(* CODESYS project test_IMA-TECHDays
   Author: SESA697794
   DefaultNamespace: MulticarrierExample
   Title: Git_example
   Version: 0.0.0.0

Project tree, tasks and I/O mapping:
  LMC_PacDrive : PacDrive LMC 300/400/402/600/802/902C, Schneider Electric, order no. LMC Pro and Pro2, version 1.76.12.4
    application Application
      libraries: PD_PacDriveLib, 1.11.1.0 (Schneider Electric); ApplicationLogger, 1.1.7.0 (Schneider Electric); Mathematics, 1.0.4.0 (Schneider Electric); Multicarrier, 1.3.6.0 (Schneider Electric); MulticarrierStation, 1.2.0.0 (Schneider Electric); DigitalTwinCommunication, 1.2.1.0 (Schneider Electric); SercosCommunication, 1.2.4.0 (Schneider Electric); PD_SoMotionGenerator, 1.9.4.0 (Schneider Electric); SysMem, * (System); SysTime, * (System); TcpUdpCommunication, 2.3.0.0 (Schneider Electric); PD_GlobalDiagnostics, 1.6.0.0 (Schneider Electric); PD_AxisModule, 1.7.1.0 (Schneider Electric); PD_Template, 1.9.0.0 (Schneider Electric); IecRtsServices, 1.0.5.0 (Schneider Electric); VisuDialogs, * (System)
      task TASK_Communication (cyclic, interval T#20ms, priority 30) calls SR_EmulationInterface, SR_OpcUa
      task TASK_SR_Diagnostics (cyclic, interval T#100ms, priority 31, watchdog T#100ms x 2) calls SR_Diagnostics
      task TASK_SR_Logging (cyclic, interval T#10ms, priority 13, watchdog T#10ms x 2) calls SR_Logging
      task TASK_SR_MainMachine (cyclic, interval T#5ms, priority 8, watchdog T#5ms x 10) calls SR_HWCopyIO, SR_MainMachine
      task TASK_SR_SlowTask (cyclic, interval T#200ms, priority 29) calls SR_ReadControlLoopParameter, SR_WriteControlLoopParameter
      task TASK_SR_VisControl (cyclic, interval T#50ms, priority 14, watchdog T#50ms x 2) calls SR_VisControl
      Application Logger
      Check_Lib/
        function CheckBounds [ST]
        function CheckDivDInt [ST]
        function CheckDivLInt [ST]
        function CheckDivLReal [ST]
        function CheckDivReal [ST]
        function CheckPointer [ST]
        function CheckRangeSigned [ST]
        function CheckRangeUnsigned [ST]
      MulticarrierConfiguration
      MulticarrierConfiguration/
        global variables GVL_MulticarrierConfiguration
        data type ST_Carrier
        data type ST_CarrierCompound
        data type ST_CarrierType
        data type ST_Part
        data type ST_PartType
        data type ST_Physics
        data type ST_ProductType
        data type ST_Segment
        data type ST_SegmentType
        data type ST_Station
        data type ST_ToolType
        data type ST_Track
      MulticarrierEmulation/
        global variables GVL_MulticarrierEmulation
        program SR_EmulationInterface [ST]: Init_MulticarrierEmulation
        Symbol Configuration
      ParameterListCarrier
      ParameterListSegments
      TemplateFullProgrammingFramework/
        CamDiagram_Slave1
          Segment
          Segment
          Segment
        CamDiagram_Slave2
          Segment
          Segment
          Segment
        EquipmentModules/
          MulticarrierModule/
            data type ET_OpModeVis
            data type ET_TraceSource
            data type ET_VisPosGapDist
            function FC_LrealEqual [ST]
            function FC_SplitString [ST]
            Multicarrier Stations/
              AutomaticMode/
                Base Station/
                  data type ET_ResultSource
                  data type ET_ResultStation
                  data type ET_StationType
                function block FB_Station1 [ST]: CyclicMotionCall
                visualisation Vis_Auto
                visualisation Vis_StationCopyMaster
              data type ST_StationParameter
              Test Multicarrier/
                01_PlayGround/
                  Traces/
                  Vis_MoveCmds/
                02_SimpleStation/
                03_PosAndSync/
                04_ColorStations/
                05_VelLimitStation/
                06_StandardStations/
                07_ExternalMaster/
                08_Superimpose/
                function block FB_MotionTestStationBase [ST]
                program SR_CallTestStations [ST]
                data type ST_CarrierMotionData
                data type ST_EmulationTestStations
                visualisation Vis_TestMulticarrier
            program SR_CarriersInStationToTrace [ST]: Call
            program SR_MulticarrierModule [SFC]: Init_CmdTables, Init_SubModules, ControlEnable, ControlModule, AddMessageToAPL, APLStartPosEndPos, TraceAndAPL, TraceStartPosEndPos, ExceptionControl_Action, HardwareFaults, Init_Exceptions, Init_Reactions, ModuleFaults, StopAllCarriers, ExitLastOpMode, MoveAllCarriersInFirstStation, SetMinGapForMoveGapControl, VirtualSetPosOfAllCarriers, Init_Carriers, Init_CrashPrevention, Init_FeedbackForVis, Init_Track, InitModule_Action, Manual_Entry, Manual_Exit, Manual_Logic, RegisterLoggerPoint, CallAllStations, DeleteAllCarriersFromStations, ErrorQuitStations, ErrorsFromStations, Init_RegisterStationsToAPL, ParameterStation1, ParameterStation2, SetStationTriggerViaTimer, TraceStations, StoreCurrentMoveCmds, Input_Action, Logger_Action, Logic_active, Output_Active, Start_Action, SubModules_Action, UpdateStructs, TrackCalibration_Logic
            data type ST_MulticarrierModule
            Traces/
              trace Trace_PosVelAcc_CurrentTrackDeviation (task SystemMotionTask): SR_MulticarrierModule.aifTraceObject[1].udiCarrierIndex, SR_MulticarrierModule.aifTraceObject[1].ifFeedbackMotionValues.lrRefTrackPosition, SR_MulticarrierModule.aifTraceObject[1].ifFeedbackMotionValues.lrRefVelocity, SR_MulticarrierModule.aifTraceObject[1].ifFeedbackMotionValues.lrRefAcceleration, SR_MulticarrierModule.aifTraceCarrierMovementData[1].ActualCurrent, SR_MulticarrierModule.aifTraceCarrierMovementData[1].TrackingDeviation, SR_MulticarrierModule.aifTraceObject[2].udiCarrierIndex, SR_MulticarrierModule.aifTraceObject[2].ifFeedbackMotionValues.lrRefTrackPosition, SR_MulticarrierModule.aifTraceObject[2].ifFeedbackMotionValues.lrRefVelocity, SR_MulticarrierModule.aifTraceObject[2].ifFeedbackMotionValues.lrRefAcceleration, SR_MulticarrierModule.aifTraceCarrierMovementData[2].ActualCurrent, SR_MulticarrierModule.aifTraceCarrierMovementData[2].TrackingDeviation, SR_MulticarrierModule.aifTraceObject[3].udiCarrierIndex, SR_MulticarrierModule.aifTraceObject[3].ifFeedbackMotionValues.lrRefTrackPosition, SR_MulticarrierModule.aifTraceObject[3].ifFeedbackMotionValues.lrRefVelocity, SR_MulticarrierModule.aifTraceObject[3].ifFeedbackMotionValues.lrRefAcceleration, SR_MulticarrierModule.aifTraceCarrierMovementData[3].ActualCurrent, SR_MulticarrierModule.aifTraceCarrierMovementData[3].TrackingDeviation, SR_MulticarrierModule.aifTraceObject[4].udiCarrierIndex, SR_MulticarrierModule.aifTraceObject[4].ifFeedbackMotionValues.lrRefTrackPosition, SR_MulticarrierModule.aifTraceObject[4].ifFeedbackMotionValues.lrRefVelocity, SR_MulticarrierModule.aifTraceObject[4].ifFeedbackMotionValues.lrRefAcceleration, SR_MulticarrierModule.aifTraceCarrierMovementData[4].ActualCurrent, SR_MulticarrierModule.aifTraceCarrierMovementData[4].TrackingDeviation, SR_MulticarrierModule.aifTraceObject[5].udiCarrierIndex, SR_MulticarrierModule.aifTraceObject[5].ifFeedbackMotionValues.lrRefTrackPosition, SR_MulticarrierModule.aifTraceObject[5].ifFeedbackMotionValues.lrRefVelocity, SR_MulticarrierModule.aifTraceObject[5].ifFeedbackMotionValues.lrRefAcceleration, SR_MulticarrierModule.aifTraceCarrierMovementData[5].ActualCurrent, SR_MulticarrierModule.aifTraceCarrierMovementData[5].TrackingDeviation
              trace Trace_PosVelAcc_Gap_InFront (task SystemMotionTask): SR_MulticarrierModule.aifTraceObject[1].udiCarrierIndex, SR_MulticarrierModule.aifTraceObject[1].ifFeedbackMotionValues.lrRefTrackPosition, SR_MulticarrierModule.aifTraceObject[1].ifFeedbackMotionValues.lrRefVelocity, SR_MulticarrierModule.aifTraceObject[1].ifFeedbackMotionValues.lrRefAcceleration, SR_MulticarrierModule.aifTraceObject[1].ifFeedbackToInFront.lrGapToCarrierInFront, SR_MulticarrierModule.aifTraceObject[2].udiCarrierIndex, SR_MulticarrierModule.aifTraceObject[2].ifFeedbackMotionValues.lrRefTrackPosition, SR_MulticarrierModule.aifTraceObject[2].ifFeedbackMotionValues.lrRefVelocity, SR_MulticarrierModule.aifTraceObject[2].ifFeedbackMotionValues.lrRefAcceleration, SR_MulticarrierModule.aifTraceObject[2].ifFeedbackToInFront.lrGapToCarrierInFront, SR_MulticarrierModule.aifTraceObject[3].udiCarrierIndex, SR_MulticarrierModule.aifTraceObject[3].ifFeedbackMotionValues.lrRefTrackPosition, SR_MulticarrierModule.aifTraceObject[3].ifFeedbackMotionValues.lrRefVelocity, SR_MulticarrierModule.aifTraceObject[3].ifFeedbackMotionValues.lrRefAcceleration, SR_MulticarrierModule.aifTraceObject[3].ifFeedbackToInFront.lrGapToCarrierInFront, SR_MulticarrierModule.aifTraceObject[4].udiCarrierIndex, SR_MulticarrierModule.aifTraceObject[4].ifFeedbackMotionValues.lrRefTrackPosition, SR_MulticarrierModule.aifTraceObject[4].ifFeedbackMotionValues.lrRefVelocity, SR_MulticarrierModule.aifTraceObject[4].ifFeedbackMotionValues.lrRefAcceleration, SR_MulticarrierModule.aifTraceObject[4].ifFeedbackToInFront.lrGapToCarrierInFront, SR_MulticarrierModule.aifTraceObject[5].udiCarrierIndex, SR_MulticarrierModule.aifTraceObject[5].ifFeedbackMotionValues.lrRefTrackPosition, SR_MulticarrierModule.aifTraceObject[5].ifFeedbackMotionValues.lrRefVelocity, SR_MulticarrierModule.aifTraceObject[5].ifFeedbackMotionValues.lrRefAcceleration, SR_MulticarrierModule.aifTraceObject[5].ifFeedbackToInFront.lrGapToCarrierInFront
              trace Trace_PosVelAcc_Gap_InFront_InTargets (task SystemMotionTask): SR_MulticarrierModule.aifTraceObject[1].udiCarrierIndex, SR_MulticarrierModule.aifTraceObject[1].ifFeedbackMotionValues.lrRefTrackPosition, SR_MulticarrierModule.aifTraceObject[1].ifFeedbackMotionValues.lrRefVelocity, SR_MulticarrierModule.aifTraceObject[1].ifFeedbackMotionValues.lrRefAcceleration, SR_MulticarrierModule.aifTraceObject[1].ifFeedbackToInFront.lrGapToCarrierInFront, SR_MulticarrierModule.aifTraceObject[1].ifFeedbackMoveGapControl.xInTemporaryTargetPosition, SR_MulticarrierModule.aifTraceObject[1].ifFeedbackMoveGapControl.xInEndTargetPosition, SR_MulticarrierModule.aifTraceObject[2].udiCarrierIndex, SR_MulticarrierModule.aifTraceObject[2].ifFeedbackMotionValues.lrRefTrackPosition, SR_MulticarrierModule.aifTraceObject[2].ifFeedbackMotionValues.lrRefVelocity, SR_MulticarrierModule.aifTraceObject[2].ifFeedbackMotionValues.lrRefAcceleration, SR_MulticarrierModule.aifTraceObject[2].ifFeedbackToInFront.lrGapToCarrierInFront, SR_MulticarrierModule.aifTraceObject[2].ifFeedbackMoveGapControl.xInTemporaryTargetPosition, SR_MulticarrierModule.aifTraceObject[2].ifFeedbackMoveGapControl.xInEndTargetPosition, SR_MulticarrierModule.aifTraceObject[3].udiCarrierIndex, SR_MulticarrierModule.aifTraceObject[3].ifFeedbackMotionValues.lrRefTrackPosition, SR_MulticarrierModule.aifTraceObject[3].ifFeedbackMotionValues.lrRefVelocity, SR_MulticarrierModule.aifTraceObject[3].ifFeedbackMotionValues.lrRefAcceleration, SR_MulticarrierModule.aifTraceObject[3].ifFeedbackToInFront.lrGapToCarrierInFront, SR_MulticarrierModule.aifTraceObject[3].ifFeedbackMoveGapControl.xInTemporaryTargetPosition, SR_MulticarrierModule.aifTraceObject[3].ifFeedbackMoveGapControl.xInEndTargetPosition, SR_MulticarrierModule.aifTraceObject[4].udiCarrierIndex, SR_MulticarrierModule.aifTraceObject[4].ifFeedbackMotionValues.lrRefTrackPosition, SR_MulticarrierModule.aifTraceObject[4].ifFeedbackMotionValues.lrRefVelocity, SR_MulticarrierModule.aifTraceObject[4].ifFeedbackMotionValues.lrRefAcceleration, SR_MulticarrierModule.aifTraceObject[4].ifFeedbackToInFront.lrGapToCarrierInFront, SR_MulticarrierModule.aifTraceObject[4].ifFeedbackMoveGapControl.xInTemporaryTargetPosition, SR_MulticarrierModule.aifTraceObject[4].ifFeedbackMoveGapControl.xInEndTargetPosition, SR_MulticarrierModule.aifTraceObject[5].udiCarrierIndex, SR_MulticarrierModule.aifTraceObject[5].ifFeedbackMotionValues.lrRefTrackPosition, SR_MulticarrierModule.aifTraceObject[5].ifFeedbackMotionValues.lrRefVelocity, SR_MulticarrierModule.aifTraceObject[5].ifFeedbackMotionValues.lrRefAcceleration, SR_MulticarrierModule.aifTraceObject[5].ifFeedbackToInFront.lrGapToCarrierInFront, SR_MulticarrierModule.aifTraceObject[5].ifFeedbackMoveGapControl.xInTemporaryTargetPosition, SR_MulticarrierModule.aifTraceObject[5].ifFeedbackMoveGapControl.xInEndTargetPosition
              trace Trace_PosVelAcc_Gap_InFront_Queued (task SystemMotionTask): SR_MulticarrierModule.aifTraceObject[1].udiCarrierIndex, SR_MulticarrierModule.aifTraceObject[1].ifFeedbackMotionValues.lrRefTrackPosition, SR_MulticarrierModule.aifTraceObject[1].ifFeedbackMotionValues.lrRefVelocity, SR_MulticarrierModule.aifTraceObject[1].ifFeedbackMotionValues.lrRefAcceleration, SR_MulticarrierModule.aifTraceObject[1].ifFeedbackToInFront.lrGapToCarrierInFront, SR_MulticarrierModule.aifTraceObject[1].ifFeedbackMoveGapControl.xQueued, SR_MulticarrierModule.aifTraceObject[1].ifFeedbackMoveGapControl.xInTemporaryTargetPosition, SR_MulticarrierModule.aifTraceObject[1].ifFeedbackMoveGapControl.xInEndTargetPosition, SR_MulticarrierModule.aifTraceObject[2].udiCarrierIndex, SR_MulticarrierModule.aifTraceObject[2].ifFeedbackMotionValues.lrRefTrackPosition, SR_MulticarrierModule.aifTraceObject[2].ifFeedbackMotionValues.lrRefVelocity, SR_MulticarrierModule.aifTraceObject[2].ifFeedbackMotionValues.lrRefAcceleration, SR_MulticarrierModule.aifTraceObject[2].ifFeedbackToInFront.lrGapToCarrierInFront, SR_MulticarrierModule.aifTraceObject[2].ifFeedbackMoveGapControl.xQueued, SR_MulticarrierModule.aifTraceObject[2].ifFeedbackMoveGapControl.xInTemporaryTargetPosition, SR_MulticarrierModule.aifTraceObject[2].ifFeedbackMoveGapControl.xInEndTargetPosition, SR_MulticarrierModule.aifTraceObject[3].udiCarrierIndex, SR_MulticarrierModule.aifTraceObject[3].ifFeedbackMotionValues.lrRefTrackPosition, SR_MulticarrierModule.aifTraceObject[3].ifFeedbackMotionValues.lrRefVelocity, SR_MulticarrierModule.aifTraceObject[3].ifFeedbackMotionValues.lrRefAcceleration, SR_MulticarrierModule.aifTraceObject[3].ifFeedbackToInFront.lrGapToCarrierInFront, SR_MulticarrierModule.aifTraceObject[3].ifFeedbackMoveGapControl.xQueued, SR_MulticarrierModule.aifTraceObject[3].ifFeedbackMoveGapControl.xInTemporaryTargetPosition, SR_MulticarrierModule.aifTraceObject[3].ifFeedbackMoveGapControl.xInEndTargetPosition, SR_MulticarrierModule.aifTraceObject[4].udiCarrierIndex, SR_MulticarrierModule.aifTraceObject[4].ifFeedbackMotionValues.lrRefTrackPosition, SR_MulticarrierModule.aifTraceObject[4].ifFeedbackMotionValues.lrRefVelocity, SR_MulticarrierModule.aifTraceObject[4].ifFeedbackMotionValues.lrRefAcceleration, SR_MulticarrierModule.aifTraceObject[4].ifFeedbackToInFront.lrGapToCarrierInFront, SR_MulticarrierModule.aifTraceObject[4].ifFeedbackMoveGapControl.xQueued, SR_MulticarrierModule.aifTraceObject[4].ifFeedbackMoveGapControl.xInTemporaryTargetPosition, SR_MulticarrierModule.aifTraceObject[4].ifFeedbackMoveGapControl.xInEndTargetPosition, SR_MulticarrierModule.aifTraceObject[5].udiCarrierIndex, SR_MulticarrierModule.aifTraceObject[5].ifFeedbackMotionValues.lrRefTrackPosition, SR_MulticarrierModule.aifTraceObject[5].ifFeedbackMotionValues.lrRefVelocity, SR_MulticarrierModule.aifTraceObject[5].ifFeedbackMotionValues.lrRefAcceleration, SR_MulticarrierModule.aifTraceObject[5].ifFeedbackToInFront.lrGapToCarrierInFront, SR_MulticarrierModule.aifTraceObject[5].ifFeedbackMoveGapControl.xQueued, SR_MulticarrierModule.aifTraceObject[5].ifFeedbackMoveGapControl.xInTemporaryTargetPosition, SR_MulticarrierModule.aifTraceObject[5].ifFeedbackMoveGapControl.xInEndTargetPosition
              trace Trace_PosVelAcc_Queued_VelocityState (task SystemMotionTask): SR_MulticarrierModule.aifTraceObject[1].udiCarrierIndex, SR_MulticarrierModule.aifTraceObject[1].ifFeedbackMotionValues.lrRefTrackPosition, SR_MulticarrierModule.aifTraceObject[1].ifFeedbackMotionValues.lrRefVelocity, SR_MulticarrierModule.aifTraceObject[1].ifFeedbackMotionValues.lrRefAcceleration, SR_MulticarrierModule.aifTraceObject[1].ifFeedbackMoveGapControl.xQueued, SR_MulticarrierModule.aifTraceObject[1].ifFeedbackMoveGapControl.etVelocityPhase, SR_MulticarrierModule.aifTraceObject[2].udiCarrierIndex, SR_MulticarrierModule.aifTraceObject[2].ifFeedbackMotionValues.lrRefTrackPosition, SR_MulticarrierModule.aifTraceObject[2].ifFeedbackMotionValues.lrRefVelocity, SR_MulticarrierModule.aifTraceObject[2].ifFeedbackMotionValues.lrRefAcceleration, SR_MulticarrierModule.aifTraceObject[2].ifFeedbackMoveGapControl.xQueued, SR_MulticarrierModule.aifTraceObject[2].ifFeedbackMoveGapControl.etVelocityPhase, SR_MulticarrierModule.aifTraceObject[3].udiCarrierIndex, SR_MulticarrierModule.aifTraceObject[3].ifFeedbackMotionValues.lrRefTrackPosition, SR_MulticarrierModule.aifTraceObject[3].ifFeedbackMotionValues.lrRefVelocity, SR_MulticarrierModule.aifTraceObject[3].ifFeedbackMotionValues.lrRefAcceleration, SR_MulticarrierModule.aifTraceObject[3].ifFeedbackMoveGapControl.xQueued, SR_MulticarrierModule.aifTraceObject[3].ifFeedbackMoveGapControl.etVelocityPhase, SR_MulticarrierModule.aifTraceObject[4].udiCarrierIndex, SR_MulticarrierModule.aifTraceObject[4].ifFeedbackMotionValues.lrRefTrackPosition, SR_MulticarrierModule.aifTraceObject[4].ifFeedbackMotionValues.lrRefVelocity, SR_MulticarrierModule.aifTraceObject[4].ifFeedbackMotionValues.lrRefAcceleration, SR_MulticarrierModule.aifTraceObject[4].ifFeedbackMoveGapControl.xQueued, SR_MulticarrierModule.aifTraceObject[4].ifFeedbackMoveGapControl.etVelocityPhase, SR_MulticarrierModule.aifTraceObject[5].udiCarrierIndex, SR_MulticarrierModule.aifTraceObject[5].ifFeedbackMotionValues.lrRefTrackPosition, SR_MulticarrierModule.aifTraceObject[5].ifFeedbackMotionValues.lrRefVelocity, SR_MulticarrierModule.aifTraceObject[5].ifFeedbackMotionValues.lrRefAcceleration, SR_MulticarrierModule.aifTraceObject[5].ifFeedbackMoveGapControl.xQueued, SR_MulticarrierModule.aifTraceObject[5].ifFeedbackMoveGapControl.etVelocityPhase
          program SR_AlphaModule [SFC]: Check_RTB, Init_Master, Init_CmdTables, Init_SubModules, ExceptionControl_Action, Init_Exceptions, Init_Reactions, ModuleFaults, RegisterLoggerPoint, InitModule_Action, Input_Action, Logger_Action, Logic_active, Output_Active, Start_Action, SubModules_Action, UpdateStructs
          program SR_BravoModule [SFC]: Check_RTB, Init_Slave1, Init_Slave2, Init_CmdTables, Init_SubModules, ExceptionControl_Action, Init_Exceptions, Init_Reactions, ModuleFaults, RegisterLoggerPoint, InitModule_Action, Input_Action, Logger_Action, Logic_active, Mode_Select, Output_Active, Start_Action, SubModules_Action, UpdateStructs
        data type ET_Cmd
        Examples/
          ExampleDiagSources/
            function block FB_ApplicationLoggerDiagSource [ST]: CancelWriting, DiagQuit, ExceptionDuringWriting, SetDiagOutputs, WriteDiagDataControl, WriteDiagDataToFile
            function block FB_ExampleTableDiagSource [ST]: CancelWriting, DiagQuit, ExceptionDuringWriting, SetDiagOutputs, WriteDiagDataControl, WriteDiagDataToFile
            function block FB_ExampleTreeDiagSource [ST]: CancelWriting, DiagQuit, ExceptionDuringWriting, SetDiagOutputs, WriteDiagDataControl, WriteDiagDataToFile
          ExampleLeafModule/
            data type ET_DiagExtExampleLeafModule
            data type ET_ExampleLeafModuleCmd
            data type ET_ExampleLeafModuleState
            data type ET_ExceptionSource
            data type ET_ModuleType
            function block FB_ExampleLeafModule [SFC]: Auto_Action, Auto_Entry, CancelException, CheckCmd, CmdControl_Action, DiagQuit, DisableAllJobs, ExceptionHandler_Action, Homing_Action, Homing_Entry, InactiveCmdExecution, Init_Action, InitHoming_Action, InitHoming_Entry, Input_Action, Logger_Action, NoOp_Entry, Output_Active, RefuseCommand, RegisterLoggerPoint, ReportException, SetInterfaces, SetOutputs, SignalSuccessfulExecution, SignalUnSuccessfulExecution
            function block FB_ExampleLeafModuleController [ST]
            function block FB_ExampleLeafModuleVisController [ST]
            function FC_EtDiagExtExampleLeafModuleToString [ST]
            function FC_EtExampleLeafModuleCmdToString [ST]
            function FC_EtExampleLeafModuleStateToString [ST]
            function FC_UpdateExampleLeafModuleAddInterfaceStruct [ST]
            data type ST_ExampleLeafModuleInterface
        GlobalVariables/
          global variables Diagnostics
          global variables ExceptionHandling
          global variables GVL_Project
          global variables HardwareInOuts
          global variables InputVariablesEpas
          global variables InputVariablesExt
          global variables IntelligentLineShaft
          global variables Logging
          global variables RestoreAxisPosition
        ProjectDiagnostics/
          data type ET_DiagExt
          data type ET_DiagExtUser
          function FC_EtDiagExtToString [ST]
          function FC_EtDiagExtUserToString [ST]
        TaskCalls/
          program SR_Diagnostics [FBD]: SetDiagnosticsWarning
          program SR_HWCopyIO [FBD]
          program SR_Logging [FBD]
          program SR_MainMachine [SFC]: Init_CmdTables, Init_SubModules, Init_Alpha, Init_Bravo, Init_MultiCarrier, ExceptionControl_Action, Init_Exceptions, Init_Reactions, MainSystemFaults, MainUserFaults, AssignCarriers, AssignSegments, CheckArraySizeOfTrackElements, CreateTrackForSimulation, SetCarrierInterfaces, SetCarrierWorkingMode, SetSegmentInterfaces, SetSegmentWorkingMode, SetTrackInterfaces, WriteGeometryOnSegments, _aBrakeReleaseStep_active, _aBrakeReleaseStep_entry, AutoStep_Action, AutoStep_Entry, AutoStop_Action, AutoStop_Entry, InitModule_Action, Input_Action, JogMachineStep_Action, JogMachineStep_Entry, Logger_Action, ManualStep_Action, ManualStep_Entry, ModeSelect_Action, Output_Action, PrepStep_Action, PrepStep_Entry, PrepStop_Action, PrepStop_Entry, Start_Action, StopBrake_Action, StopBrake_Entry, StopJog_Action, StopJog_Entry, StopMan_Action, StopMan_Entry, StopTrackCalibration_Action, StopTrackCalibration_Entry, SubModules_Action, TestMulticarrierStep_Action, TestMulticarrierStep_Entry, TestMulticarrierStop_Action, TestMulticarrierStop_Entry, TrackCalibrationStep_Action, TrackCalibrationStep_Entry, UpdateStructs
          program SR_OpcUa [ST]
          program SR_ReadControlLoopParameter [ST]: GetParameter, ReadParameter, SercosReadServiceDataFromSegments
          program SR_VisControl [ST]: CallTestErrors, CurrentModuleCmdTable, DetectOpModeChange, ExceptionVis, InitTestExceptions, LoggerVis, MainPageCmdTable, ModuleNavigationIn, ModuleNavigationOut, ModuleReaction, ModuleVisController, OpModeControl, SearchCurrentModule, SetCurrentModule
          program SR_WriteControlLoopParameter [ST]: SercosWriteServiceDataToAllSegments, StartAndSetParameter
        Tools/
          function FC_IsDriveVirtual [ST]
          function FC_ObjectTypeIsMotionAxis [ST]
          function FC_SetDeadTimeCompensation [ST]
          Multicarrier/
        Visualization/
          Examples/
            visualisation FR_ButtonAssignId
            visualisation FR_ExampleLeafModule
            visualisation FR_ExampleLeafModuleSelect
            visualisation VIS_ExampleLeafModule
          FramesProject/
            visualisation FR_ControlModuleTypes
            visualisation FR_NavigationButtons
            visualisation FR_OtherModuleTypes
          Multicarrier/
            visualisation FR_CarDist
            visualisation FR_List
            text list TextList_VisPositions
            visualisation Vis_ApplicationLogger
            visualisation Vis_Error
            visualisation Vis_Jogging
            visualisation Vis_NoOpMode
            visualisation Vis_Positions
            visualisation Vis_Positions_121_150
            visualisation Vis_Positions_1_30
            visualisation Vis_Positions_31_60
            visualisation Vis_Positions_61_90
            visualisation Vis_Positions_91_120
            visualisation Vis_Trace
            visualisation Vis_TrackCalibration
          visualisation VIS_Main
          visualisation Vis_Multicarrier
          Windows/
            visualisation VIS_AxisModule
            visualisation VIS_ControlModule
            visualisation VIS_ExceptionDetails
            visualisation VIS_ExceptionList
            visualisation VIS_LogDataList
            visualisation VIS_LogDataListExt
            visualisation VIS_ModuleDetails
            visualisation VIS_ModuleExceptions
            visualisation VIS_Modules
            visualisation VIS_VisNavigation
    Device Addressing
    Message Logger
    AI_0 : Analog Input, Schneider Electric, version 1.76.12.4
    AI_1 : Analog Input, Schneider Electric, version 1.76.12.4
    AQ_0 : Analog Output, Schneider Electric, version 1.76.12.4
    AQ_1 : Analog Output, Schneider Electric, version 1.76.12.4
    DIG_DigitalIn : Digital Inputs, Schneider Electric, version 1.76.12.4
      DI_0 : Input, Schneider Electric, version 1.76.12.4
      DI_10 : Input, Schneider Electric, version 1.76.12.4
      DI_11 : Input, Schneider Electric, version 1.76.12.4
      DI_12 : Input, Schneider Electric, version 1.76.12.4
      DI_13 : Input, Schneider Electric, version 1.76.12.4
      DI_14 : Input, Schneider Electric, version 1.76.12.4
      DI_15 : Input, Schneider Electric, version 1.76.12.4
      DI_16 : Input, Schneider Electric, version 1.76.12.4
      DI_17 : Input, Schneider Electric, version 1.76.12.4
      DI_18 : Input, Schneider Electric, version 1.76.12.4
      DI_19 : Input, Schneider Electric, version 1.76.12.4
      DI_1 : Input, Schneider Electric, version 1.76.12.4
      DI_2 : Input, Schneider Electric, version 1.76.12.4
      DI_3 : Input, Schneider Electric, version 1.76.12.4
      DI_4 : Input, Schneider Electric, version 1.76.12.4
      DI_5 : Input, Schneider Electric, version 1.76.12.4
      DI_6 : Input, Schneider Electric, version 1.76.12.4
      DI_7 : Input, Schneider Electric, version 1.76.12.4
      DI_8 : Input, Schneider Electric, version 1.76.12.4
      DI_9 : Input, Schneider Electric, version 1.76.12.4
      FI_0 : Fast Input, Schneider Electric, version 1.76.12.4
      FI_1 : Fast Input, Schneider Electric, version 1.76.12.4
      FI_2 : Fast Input, Schneider Electric, version 1.76.12.4
      FI_3 : Fast Input, Schneider Electric, version 1.76.12.4
    DQG_DigitalOut : Digital Outputs, Schneider Electric, version 1.76.12.4
        settings: DiagMask = 0; OpenloadDiagMsk = 0
      DQ_0 : Output, Schneider Electric, version 1.76.12.4
      DQ_10 : Output, Schneider Electric, version 1.76.12.4
      DQ_11 : Output, Schneider Electric, version 1.76.12.4
      DQ_12 : Output, Schneider Electric, version 1.76.12.4
      DQ_13 : Output, Schneider Electric, version 1.76.12.4
      DQ_14 : Output, Schneider Electric, version 1.76.12.4
      DQ_15 : Output, Schneider Electric, version 1.76.12.4
      DQ_1 : Output, Schneider Electric, version 1.76.12.4
      DQ_2 : Output, Schneider Electric, version 1.76.12.4
      DQ_3 : Output, Schneider Electric, version 1.76.12.4
      DQ_4 : Output, Schneider Electric, version 1.76.12.4
      DQ_5 : Output, Schneider Electric, version 1.76.12.4
      DQ_6 : Output, Schneider Electric, version 1.76.12.4
      DQ_7 : Output, Schneider Electric, version 1.76.12.4
      DQ_8 : Output, Schneider Electric, version 1.76.12.4
      DQ_9 : Output, Schneider Electric, version 1.76.12.4
    LE_Master : Log. Encoder, Schneider Electric, version 1.76.12.4
    LE_Slave1 : Log. Encoder, Schneider Electric, version 1.76.12.4
    LE_Slave2 : Log. Encoder, Schneider Electric, version 1.76.12.4
    MC_CarrierPool : Lexium MC Carrier Pool, Schneider Electric, version 1.76.12.4
      MC_Carrier_10 : Lexium MC Carrier, Schneider Electric, version 1.76.12.4
      MC_Carrier_11 : Lexium MC Carrier, Schneider Electric, version 1.76.12.4
      MC_Carrier_12 : Lexium MC Carrier, Schneider Electric, version 1.76.12.4
      MC_Carrier_13 : Lexium MC Carrier, Schneider Electric, version 1.76.12.4
      MC_Carrier_14 : Lexium MC Carrier, Schneider Electric, version 1.76.12.4
      MC_Carrier_15 : Lexium MC Carrier, Schneider Electric, version 1.76.12.4
      MC_Carrier_16 : Lexium MC Carrier, Schneider Electric, version 1.76.12.4
      MC_Carrier_17 : Lexium MC Carrier, Schneider Electric, version 1.76.12.4
      MC_Carrier_18 : Lexium MC Carrier, Schneider Electric, version 1.76.12.4
      MC_Carrier_19 : Lexium MC Carrier, Schneider Electric, version 1.76.12.4
      MC_Carrier_1 : Lexium MC Carrier, Schneider Electric, version 1.76.12.4
      MC_Carrier_20 : Lexium MC Carrier, Schneider Electric, version 1.76.12.4
      MC_Carrier_21 : Lexium MC Carrier, Schneider Electric, version 1.76.12.4
      MC_Carrier_22 : Lexium MC Carrier, Schneider Electric, version 1.76.12.4
      MC_Carrier_23 : Lexium MC Carrier, Schneider Electric, version 1.76.12.4
      MC_Carrier_24 : Lexium MC Carrier, Schneider Electric, version 1.76.12.4
      MC_Carrier_25 : Lexium MC Carrier, Schneider Electric, version 1.76.12.4
      MC_Carrier_26 : Lexium MC Carrier, Schneider Electric, version 1.76.12.4
      MC_Carrier_27 : Lexium MC Carrier, Schneider Electric, version 1.76.12.4
      MC_Carrier_28 : Lexium MC Carrier, Schneider Electric, version 1.76.12.4
      MC_Carrier_29 : Lexium MC Carrier, Schneider Electric, version 1.76.12.4
      MC_Carrier_2 : Lexium MC Carrier, Schneider Electric, version 1.76.12.4
      MC_Carrier_30 : Lexium MC Carrier, Schneider Electric, version 1.76.12.4
      MC_Carrier_31 : Lexium MC Carrier, Schneider Electric, version 1.76.12.4
      MC_Carrier_32 : Lexium MC Carrier, Schneider Electric, version 1.76.12.4
      MC_Carrier_33 : Lexium MC Carrier, Schneider Electric, version 1.76.12.4
      MC_Carrier_34 : Lexium MC Carrier, Schneider Electric, version 1.76.12.4
      MC_Carrier_35 : Lexium MC Carrier, Schneider Electric, version 1.76.12.4
      MC_Carrier_36 : Lexium MC Carrier, Schneider Electric, version 1.76.12.4
      MC_Carrier_37 : Lexium MC Carrier, Schneider Electric, version 1.76.12.4
      MC_Carrier_38 : Lexium MC Carrier, Schneider Electric, version 1.76.12.4
      MC_Carrier_39 : Lexium MC Carrier, Schneider Electric, version 1.76.12.4
      MC_Carrier_3 : Lexium MC Carrier, Schneider Electric, version 1.76.12.4
      MC_Carrier_40 : Lexium MC Carrier, Schneider Electric, version 1.76.12.4
      MC_Carrier_41 : Lexium MC Carrier, Schneider Electric, version 1.76.12.4
      MC_Carrier_42 : Lexium MC Carrier, Schneider Electric, version 1.76.12.4
      MC_Carrier_43 : Lexium MC Carrier, Schneider Electric, version 1.76.12.4
      MC_Carrier_44 : Lexium MC Carrier, Schneider Electric, version 1.76.12.4
      MC_Carrier_45 : Lexium MC Carrier, Schneider Electric, version 1.76.12.4
      MC_Carrier_46 : Lexium MC Carrier, Schneider Electric, version 1.76.12.4
      MC_Carrier_47 : Lexium MC Carrier, Schneider Electric, version 1.76.12.4
      MC_Carrier_48 : Lexium MC Carrier, Schneider Electric, version 1.76.12.4
      MC_Carrier_49 : Lexium MC Carrier, Schneider Electric, version 1.76.12.4
      MC_Carrier_4 : Lexium MC Carrier, Schneider Electric, version 1.76.12.4
      MC_Carrier_50 : Lexium MC Carrier, Schneider Electric, version 1.76.12.4
      MC_Carrier_51 : Lexium MC Carrier, Schneider Electric, version 1.76.12.4
      MC_Carrier_52 : Lexium MC Carrier, Schneider Electric, version 1.76.12.4
      MC_Carrier_53 : Lexium MC Carrier, Schneider Electric, version 1.76.12.4
      MC_Carrier_54 : Lexium MC Carrier, Schneider Electric, version 1.76.12.4
      MC_Carrier_55 : Lexium MC Carrier, Schneider Electric, version 1.76.12.4
      MC_Carrier_56 : Lexium MC Carrier, Schneider Electric, version 1.76.12.4
      MC_Carrier_57 : Lexium MC Carrier, Schneider Electric, version 1.76.12.4
      MC_Carrier_58 : Lexium MC Carrier, Schneider Electric, version 1.76.12.4
      MC_Carrier_59 : Lexium MC Carrier, Schneider Electric, version 1.76.12.4
      MC_Carrier_5 : Lexium MC Carrier, Schneider Electric, version 1.76.12.4
      MC_Carrier_60 : Lexium MC Carrier, Schneider Electric, version 1.76.12.4
      MC_Carrier_61 : Lexium MC Carrier, Schneider Electric, version 1.76.12.4
      MC_Carrier_62 : Lexium MC Carrier, Schneider Electric, version 1.76.12.4
      MC_Carrier_63 : Lexium MC Carrier, Schneider Electric, version 1.76.12.4
      MC_Carrier_64 : Lexium MC Carrier, Schneider Electric, version 1.76.12.4
      MC_Carrier_65 : Lexium MC Carrier, Schneider Electric, version 1.76.12.4
      MC_Carrier_66 : Lexium MC Carrier, Schneider Electric, version 1.76.12.4
      MC_Carrier_67 : Lexium MC Carrier, Schneider Electric, version 1.76.12.4
      MC_Carrier_68 : Lexium MC Carrier, Schneider Electric, version 1.76.12.4
      MC_Carrier_69 : Lexium MC Carrier, Schneider Electric, version 1.76.12.4
      MC_Carrier_6 : Lexium MC Carrier, Schneider Electric, version 1.76.12.4
      MC_Carrier_70 : Lexium MC Carrier, Schneider Electric, version 1.76.12.4
      MC_Carrier_7 : Lexium MC Carrier, Schneider Electric, version 1.76.12.4
      MC_Carrier_8 : Lexium MC Carrier, Schneider Electric, version 1.76.12.4
      MC_Carrier_9 : Lexium MC Carrier, Schneider Electric, version 1.76.12.4
    Sercos_Master : Sercos Master, Schneider Electric, version 1.76.12.4
      DRV_Master : Lexium LXM62 Drive, Schneider Electric, order no. LXM62DU60, LXM62DD15, LXM62DD27, LXM62DD45, LXM62DC13, version 1.76.12.4
      DRV_Slave1 : Lexium LXM62 Drive, Schneider Electric, order no. LXM62DU60, LXM62DD15, LXM62DD27, LXM62DD45, LXM62DC13, version 1.76.12.4
      DRV_Slave2 : Lexium LXM62 Drive, Schneider Electric, order no. LXM62DU60, LXM62DD15, LXM62DD27, LXM62DD45, LXM62DC13, version 1.76.12.4
      MC_Track_1 : Lexium MC Track, Schneider Electric, version 1.76.12.4
        MC_Segment_10 : Lexium MC Segment, Schneider Electric, version 1.76.12.4
        MC_Segment_11 : Lexium MC Segment, Schneider Electric, version 1.76.12.4
        MC_Segment_12 : Lexium MC Segment, Schneider Electric, version 1.76.12.4
            settings: ConfiguredAngleFractionNumerator = 1
        MC_Segment_13 : Lexium MC Segment, Schneider Electric, version 1.76.12.4
            settings: ConfiguredAngleFractionNumerator = 1
        MC_Segment_14 : Lexium MC Segment, Schneider Electric, version 1.76.12.4
            settings: ConfiguredAngleFractionNumerator = 1
        MC_Segment_15 : Lexium MC Segment, Schneider Electric, version 1.76.12.4
            settings: ConfiguredAngleFractionNumerator = 1
        MC_Segment_16 : Lexium MC Segment, Schneider Electric, version 1.76.12.4
        MC_Segment_17 : Lexium MC Segment, Schneider Electric, version 1.76.12.4
        MC_Segment_18 : Lexium MC Segment, Schneider Electric, version 1.76.12.4
        MC_Segment_19 : Lexium MC Segment, Schneider Electric, version 1.76.12.4
        MC_Segment_1 : Lexium MC Segment, Schneider Electric, version 1.76.12.4
        MC_Segment_20 : Lexium MC Segment, Schneider Electric, version 1.76.12.4
        MC_Segment_21 : Lexium MC Segment, Schneider Electric, version 1.76.12.4
        MC_Segment_22 : Lexium MC Segment, Schneider Electric, version 1.76.12.4
        MC_Segment_23 : Lexium MC Segment, Schneider Electric, version 1.76.12.4
        MC_Segment_24 : Lexium MC Segment, Schneider Electric, version 1.76.12.4
        MC_Segment_25 : Lexium MC Segment, Schneider Electric, version 1.76.12.4
        MC_Segment_26 : Lexium MC Segment, Schneider Electric, version 1.76.12.4
        MC_Segment_27 : Lexium MC Segment, Schneider Electric, version 1.76.12.4
            settings: ConfiguredAngleFractionNumerator = 1
        MC_Segment_28 : Lexium MC Segment, Schneider Electric, version 1.76.12.4
            settings: ConfiguredAngleFractionNumerator = 1
        MC_Segment_29 : Lexium MC Segment, Schneider Electric, version 1.76.12.4
            settings: ConfiguredAngleFractionNumerator = 1
        MC_Segment_2 : Lexium MC Segment, Schneider Electric, version 1.76.12.4
        MC_Segment_30 : Lexium MC Segment, Schneider Electric, version 1.76.12.4
            settings: ConfiguredAngleFractionNumerator = 1
        MC_Segment_3 : Lexium MC Segment, Schneider Electric, version 1.76.12.4
        MC_Segment_4 : Lexium MC Segment, Schneider Electric, version 1.76.12.4
        MC_Segment_5 : Lexium MC Segment, Schneider Electric, version 1.76.12.4
        MC_Segment_6 : Lexium MC Segment, Schneider Electric, version 1.76.12.4
        MC_Segment_7 : Lexium MC Segment, Schneider Electric, version 1.76.12.4
        MC_Segment_8 : Lexium MC Segment, Schneider Electric, version 1.76.12.4
        MC_Segment_9 : Lexium MC Segment, Schneider Electric, version 1.76.12.4
      PSM_PowerSupply : Lexium LXM62 Power Supply, Schneider Electric, order no. LXM62PD84, LXM62PD20, version 1.76.12.4
    TPG_TPIn : Touch Probe Inputs, Schneider Electric, version 1.76.12.4
      TP_0 : Touch Probe Input, Schneider Electric, version 1.76.12.4
      TP_10 : Touch Probe Input, Schneider Electric, version 1.76.12.4
      TP_11 : Touch Probe Input, Schneider Electric, version 1.76.12.4
      TP_12 : Touch Probe Input, Schneider Electric, version 1.76.12.4
      TP_13 : Touch Probe Input, Schneider Electric, version 1.76.12.4
      TP_14 : Touch Probe Input, Schneider Electric, version 1.76.12.4
      TP_15 : Touch Probe Input, Schneider Electric, version 1.76.12.4
      TP_1 : Touch Probe Input, Schneider Electric, version 1.76.12.4
      TP_2 : Touch Probe Input, Schneider Electric, version 1.76.12.4
      TP_3 : Touch Probe Input, Schneider Electric, version 1.76.12.4
      TP_4 : Touch Probe Input, Schneider Electric, version 1.76.12.4
      TP_5 : Touch Probe Input, Schneider Electric, version 1.76.12.4
      TP_6 : Touch Probe Input, Schneider Electric, version 1.76.12.4
      TP_7 : Touch Probe Input, Schneider Electric, version 1.76.12.4
      TP_8 : Touch Probe Input, Schneider Electric, version 1.76.12.4
      TP_9 : Touch Probe Input, Schneider Electric, version 1.76.12.4
  00000000-0000-0000-0000-000000000000|M:\lib-jenkins-config\externalfiles\Disclaimer of Warranty.pdf
  Disclaimer of Warranty
  text list GlobalTextList
  Project Information/
    function GetBooleanProperty [ST]
    function GetCompany [ST]
    function GetNumberProperty [ST]
    function GetTextProperty2 [ST]
    function GetTextProperty [ST]
    function GetTitle [ST]
    function GetVersion [ST]
    function GetVersionProperty [ST]
*)

// LMC_PacDrive/Application/MulticarrierConfiguration/ST_Carrier
// generated content, do not modify
TYPE ST_Carrier :
STRUCT
	diCarrierCompoundsIndex : DINT;
END_STRUCT
END_TYPE

// LMC_PacDrive/Application/MulticarrierConfiguration/ST_CarrierCompound
// generated content, do not modify
TYPE ST_CarrierCompound :
STRUCT
	sName : STRING;
	sDescription : STRING;
	stCarrierType : STRING;
	stToolOffset : SE_MATH.ST_Vector3D;
	stProductOffset : SE_MATH.ST_Vector3D;
	diToolTypesIndex : DINT;
END_STRUCT
END_TYPE

// LMC_PacDrive/Application/MulticarrierConfiguration/ST_CarrierType
// generated content, do not modify
TYPE ST_CarrierType :
STRUCT
	sName: STRING;
	sDescription: STRING;
	stPhysics: ST_Physics;
	stToolOffset: SE_MATH.ST_Vector3D;
	iToolOffsetBase: INT;
	diToolTypesIndex: DINT;
END_STRUCT
END_TYPE

// LMC_PacDrive/Application/MulticarrierConfiguration/ST_Part
// generated content, do not modify
TYPE ST_Part :
STRUCT
	stLocation : SE_MATH.ST_Vector3D;
	diPartTypesIndex : DINT;
END_STRUCT
END_TYPE

// LMC_PacDrive/Application/MulticarrierConfiguration/ST_PartType
// generated content, do not modify
TYPE ST_PartType :
STRUCT
	lrHeight : LREAL;
	sPoints : STRING;
END_STRUCT
END_TYPE

// LMC_PacDrive/Application/MulticarrierConfiguration/ST_Physics
// generated content, do not modify
TYPE ST_Physics :
STRUCT
	stDimensions : MCR.ST_Dimensions;
END_STRUCT
END_TYPE

// LMC_PacDrive/Application/MulticarrierConfiguration/ST_ProductType
// generated content, do not modify
TYPE ST_ProductType :
STRUCT
	sName : STRING;
	sDescription : STRING;
	stPhysics : ST_Physics;
END_STRUCT
END_TYPE

// LMC_PacDrive/Application/MulticarrierConfiguration/ST_Segment
// generated content, do not modify
TYPE ST_Segment :
STRUCT
	diSegmentTypesIndex : DINT;
END_STRUCT
END_TYPE

// LMC_PacDrive/Application/MulticarrierConfiguration/ST_SegmentType
// generated content, do not modify
TYPE ST_SegmentType :
STRUCT
	lrRailLength : LREAL;
	xIsCurved : BOOL;
	lrAngle : LREAL;
	diAngleFractionNumerator : DINT;
	udiAngleFractionDenominator : UDINT;
END_STRUCT
END_TYPE

// LMC_PacDrive/Application/MulticarrierConfiguration/ST_Station
// generated content, do not modify
TYPE ST_Station :
STRUCT
	sName : STRING;
	lrWaitPosition : LREAL;
	lrProcessPosition : LREAL;
END_STRUCT
END_TYPE

// LMC_PacDrive/Application/MulticarrierConfiguration/ST_ToolType
// generated content, do not modify
TYPE ST_ToolType :
STRUCT
	sName : STRING;
	sDescription : STRING;
	stPhysics : ST_Physics;
	sPartsIndices : STRING;
END_STRUCT
END_TYPE

// LMC_PacDrive/Application/MulticarrierConfiguration/ST_Track
// generated content, do not modify
TYPE ST_Track :
STRUCT
	xIsClosed : BOOL;
	xDirection : BOOL;
	lrLength : LREAL;
	lrLogicalStartOffset : LREAL;
	udiNumberOfSegments : UDINT;
	astSegments : ARRAY [1..GVL_MulticarrierConfiguration.Gc_udiMaxNumberOfSegments] OF ST_Segment;
	udiNumberOfStations : UDINT;
	astStations : ARRAY [1..GVL_MulticarrierConfiguration.Gc_udiMaxNumberOfStations] OF ST_Station;
END_STRUCT
END_TYPE

// LMC_PacDrive/Application/TemplateFullProgrammingFramework/ET_Cmd
{attribute 'qualified_only'}
TYPE ET_Cmd :
(	NoCmd				:= 0,

	(* TPL.Gc_udiUserCmdOffset : UDINT := 25000; // >= 25000: user defined Commands *)
	DriveEnableOn		:= 25999,
	DriveEnableOff		:= 25998,
	Init				:= 25997,
	Prepare				:= 25996,
	Production			:= 25995,
	Auto				:= 25994,
	BrakeRelease		:= 25993,
	Abort				:= 25992,
	Standby				:= 25991,
	Manual				:= 25990,
	Jogging				:= 25989,
	Hold				:= 25988,
	Stop				:= 25987,
	Start				:= 25986,
	HoldJM				:= 25985,
	TestMulticarrier	:= 25984,
	StopPrepare			:= 25983,
	StopAuto			:= 25982,
	TrackCalibration	:= 25981
)DINT;
END_TYPE

// LMC_PacDrive/Application/TemplateFullProgrammingFramework/ProjectDiagnostics/ET_DiagExt
{attribute 'qualified_only'}
TYPE ET_DiagExt :
(
	(* Minimum value +0 *)
	Ok								:= 0,
	Disabled						:= 1,
	WaitUntilControllerFinishedBoot	:= 2,
	Initializing					:= 3,
	DeactivatingSubModules			:= 4,
	ExecuteStep						:= 5,
	WaitAtNegativeStep				:= 6,
	WaitCmdsDone					:= 7,
	WaitForCmd						:= 8,
	SubModuleInException			:= 9,
	ModuleControllerException		:= 10,
	UnknownStateModuleController	:= 11,
	
	SystemFatalException			:= 12,
	SystemException					:= 13,
	SystemWarning					:= 14,
	MainSystemEmergencyStop			:= 15,
	InvalidPointer					:= 16,	
	UpdateStructsException			:= 17,
	InitReactionsException			:= 18,
	InitSubModulesException			:= 19,
	ifMulticarrierSegmentsInvalid 	:= 20,
	UnknownDiagExt					:= 21,
	
	Exception1FromVis				:= 22,
	Exception2FromVis				:= 23,
	Exception3FromVis				:= 24,
	Exception4FromVis				:= 25,
	Exception5FromVis				:= 26,
	
	DiagnosticsWarning					:= 27,
	WaitUntilDiagnosticsManagerReady	:= 28,
	WaitUntilDisabled					:= 29,
	WaitUntilDiagSourceRegistered		:= 30,
	WaitForCommunication				:= 31,
	DataSuccessfullyWritten				:= 32,
	WritingToFile						:= 33,
	FileIdInvalid						:= 34,
	CmdUnknown							:= 35,	

	WaitUntilSercosState4				:= 36,

	UnexpectedFeedback					:= 37,
	UnknownDiagExtUser					:= 38,
	HardwareException					:= 39,
	InvalidConfiguredParameter			:= 40,
	TimeoutControlEnable				:= 41,
	SegmentNotEnabled					:= 42

)UDINT;
END_TYPE

// LMC_PacDrive/Application/TemplateFullProgrammingFramework/ProjectDiagnostics/ET_DiagExtUser
{attribute 'qualified_only'}
TYPE ET_DiagExtUser :
(
(* Minimum value +0 *)
	Exception1FromEquipmentModule		:= 0,
	Exception2FromEquipmentModule		:= 1,
	
	Exception1FromMain					:= 2,
	Exception2FromMain					:= 3,
	Exception3FromMain					:= 4,
	Exception4FromMain					:= 5,
	Exception5FromMain					:= 6
	
	
	
)UDINT;
END_TYPE

// LMC_PacDrive/Application/TemplateFullProgrammingFramework/EquipmentModules/MulticarrierModule/ET_OpModeVis
{attribute 'qualified_only'}
{attribute 'strict'}
TYPE ET_OpModeVis :
(
	None,Manual,Auto,Test,TrackCalibration
)UINT;
END_TYPE

// LMC_PacDrive/Application/TemplateFullProgrammingFramework/EquipmentModules/MulticarrierModule/ET_TraceSource
{attribute 'qualified_only'}
{attribute 'strict'}
TYPE ET_TraceSource :
(
	MulticarrierModule,
	Station1,
	Station2,
	Station3,
	Station4,
	Station5,
	Station6,
	Station7,
	Station8,
	Station9,
	Station10,
	Station11,
	Station12,
	Station13,
	Station14,
	Station15,
	Station16,
	Station17,
	Station18,
	Station19,
	Station20,
	Station21,
	Station22,
	Station23,
	Station24,
	Station25,
	Station26,
	Station27,
	Station28,
	Station29,
	Station30,
	LoadTestMulticarrier,
	UnLoadTestMulticarrier,
	LoadPlayGround,
	UnLoadPlayGround,
	LoadSimple,
	FillSmple,
	UnLoadSimple,
	LoadPosAndSync,
	FillPosAndSync,
	ClosePosandSync,
	UnLoadPosAndSync,
	LoadColor,
	RedColor,
	BlueColor,
	YellowColor,
	UnloadColor,
	VelLimitStation1,
	VelLimitStation2,
	AutoStation1,
	ClampingStation,
	DeclampingStation,
	GroupStation1,
	GroupStation2,
	SyncToExternalMaster,
	WaitLoad,
	LoadAndSuperimposeClamping,
	SuperimposeDeclampAndUnload,
	StartPosAndEndPos
);
END_TYPE

// LMC_PacDrive/Application/TemplateFullProgrammingFramework/EquipmentModules/MulticarrierModule/ET_VisPosGapDist
{attribute 'qualified_only'}
{attribute 'strict'}
TYPE ET_VisPosGapDist :
(
	RefTrackPosition,
	RefPosition,
	GapToCarrierInFront,
	DistanceToCarrierInFront,
	GapToCarrierBehind,
	DistanceToCarrierBehind
);
END_TYPE

// LMC_PacDrive/Application/TemplateFullProgrammingFramework/EquipmentModules/MulticarrierModule/ST_MulticarrierModule
TYPE ST_MulticarrierModule :
STRUCT
	//-- Arrays filled in SR_MainMachine.Start_Action	
	i_ifMulticarrierTrack				: SystemConfigurationItf.IF_MulticarrierTrack;
	i_ifMulticarrierTrackEnableAccess	: SystemUserFunctionsItf.IF_TrackEnableAccess;
	i_ifMulticarrierTrackEnable			: SystemUserFunctionsItf.IF_TrackEnable;
	i_aifIdentificationMandatory		: ARRAY[1..MCR.GPL.Gc_udiMaxNumberOfCarriers] OF SystemConfigurationItf.IF_IdentificationMandatory;
	i_aifMulticarrierCarriers			: ARRAY[1..MCR.GPL.Gc_udiMaxNumberOfCarriers] OF SystemConfigurationItf.IF_MulticarrierCarrier;
	i_aifMovementDataAccess				: ARRAY[1..MCR.GPL.Gc_udiMaxNumberOfCarriers] OF SystemUserFunctionsItf.IF_MovementDataAccess;
	i_aifMovementData					: ARRAY[1..MCR.GPL.Gc_udiMaxNumberOfCarriers] OF SystemUserFunctionsItf.IF_MovementData;
	i_aifCarrierIdentificationAccess	: ARRAY[1..MCR.GPL.Gc_udiMaxNumberOfCarriers] OF SystemUserFunctionsItf.IF_CarrierIdentificationAccess;
	i_aifCarrierIdentification			: ARRAY[1..MCR.GPL.Gc_udiMaxNumberOfCarriers] OF SystemUserFunctionsItf.IF_CarrierIdentification;
	i_aifCarrierStateAccess				: ARRAY[1..MCR.GPL.Gc_udiMaxNumberOfCarriers] OF SystemUserFunctionsItf.IF_CarrierStateAccess;
	i_aifCarrierState					: ARRAY[1..MCR.GPL.Gc_udiMaxNumberOfCarriers] OF SystemUserFunctionsItf.IF_CarrierState;
	i_aifSegmentEnableAccess			: ARRAY[1..MCR.GPL.Gc_udiMaxNumberOfSegments] OF SystemUserFunctionsItf.IF_SegmentEnableAccess;
	i_aifSegmentEnable					: ARRAY[1..MCR.GPL.Gc_udiMaxNumberOfSegments] OF SystemUserFunctionsItf.IF_SegmentEnable;
	i_aifSegmentGeometryAccess			: ARRAY[1..MCR.GPL.Gc_udiMaxNumberOfSegments] OF SystemUserFunctionsItf.IF_SegmentGeometryAccess;
	i_aifSegmentGeometry				: ARRAY[1..MCR.GPL.Gc_udiMaxNumberOfSegments] OF SystemUserFunctionsItf.IF_SegmentGeometry;
	
	i_aifSegmentSercosIdentificationAccess	: ARRAY[1..MCR.GPL.Gc_udiMaxNumberOfSegments] OF SystemUserFunctionsItf.IF_SercosIdentificationAccess;
	i_aifSegmentSercosIdentification		: ARRAY[1..MCR.GPL.Gc_udiMaxNumberOfSegments] OF SystemUserFunctionsItf.IF_SercosIdentification;
	i_aifMulticarrierSegments				: ARRAY[1..MCR.GPL.Gc_udiMaxNumberOfSegments] OF SystemConfigurationItf.IF_MulticarrierSegment;
	iq_xDoVirtualSetposAfterFirstProgramCall: BOOL;
END_STRUCT
END_TYPE

// LMC_PacDrive/Application/TemplateFullProgrammingFramework/Examples/ExampleLeafModule/ET_DiagExtExampleLeafModule
{attribute 'qualified_only'}
TYPE ET_DiagExtExampleLeafModule :
(
(* Minimum value +0 *)
	Ok										:= 0,
	Disabled								:= 1,
	Initializing							:= 2,
	NoOp									:= 3,
	HomingWaitForStart						:= 4,
	HomingExecuting							:= 5,
	HomingDone								:= 6,
	AutoWaitForStart						:= 7,
	AutoRunning								:= 8,
	Working									:= 9,

	UnknownDiagExtExampleLeafModule			:= 10,
	SubModuleAddInterfacesInvalidPointer	:= 11,
	SubModuleConstantRange					:= 12,
	MissingExtInit							:= 13,
	ReactionOffsetRange						:= 14,
	DriveInvalid							:= 15,
	
	CmdUnknown								:= 16,
	CmdImpossibleOverwrite					:= 17,
	CmdImpossibleState						:= 18,
	CmdImpossibleReaction					:= 19,
	
	AsyncStop								:= 20,
	SyncStopEL								:= 21,
	SyncStopEH								:= 22,
	StopEndOfCycle							:= 23,
	
	DriveFatalException						:= 24,
	DriveException							:= 25,
	DriveWarning							:= 26,
	
	UnknownState							:= 27,
	UnknownCmd								:= 28,
	RandomException							:= 29,
	
	CurrentStandardItfInvalidPointer		:= 30,
	CurrentAddItfInvalidPointer				:= 31,
	
	ParentInvalid							:= 32,
	ParentNotRegistered						:= 33,
	MaxNumberOfLoggerPointsExeeded			:= 34,
	UnexpectedDiagExt						:= 35
)UDINT;
END_TYPE

// LMC_PacDrive/Application/TemplateFullProgrammingFramework/Examples/ExampleLeafModule/ET_ExampleLeafModuleCmd
{attribute 'qualified_only'}
TYPE ET_ExampleLeafModuleCmd :
(
	(* TPL.Gc_udiUserCmdOffset : UDINT := 25000; // >= 25000: user defined Commands *)
	Homing				:= 30000,
	Auto				:= 30001,
	Start				:= 30002,
	Stop				:= 30003,
	Hold				:= 30004
	
)DINT;
END_TYPE

// LMC_PacDrive/Application/TemplateFullProgrammingFramework/Examples/ExampleLeafModule/ET_ExampleLeafModuleState
{attribute 'qualified_only'}
TYPE ET_ExampleLeafModuleState :
(
	NoOp				:= 0,
	Disabled			:= 1,
	Initializing		:= 2,
	HomingWaitForStart	:= 3,
	HomingExecuting		:= 4,
	HomingDone			:= 5,
	AutoWaitForStart	:= 6,
	AutoRunning			:= 7
)UDINT;
END_TYPE

// LMC_PacDrive/Application/TemplateFullProgrammingFramework/Examples/ExampleLeafModule/ET_ExceptionSource
{attribute 'qualified_only'}
TYPE ET_ExceptionSource :
(
	(* 0 - 9999 = reserved area *)
	
	(* Sources > 9999 = free Area *)
	ExampleLeafModule	:= 15000
)UDINT;
END_TYPE

// LMC_PacDrive/Application/TemplateFullProgrammingFramework/Examples/ExampleLeafModule/ET_ModuleType
{attribute 'qualified_only'}
TYPE ET_ModuleType :
(
	(* 0 - 9999 = reserved area *)
	(* IDs >9999 = free Area *)
	ExampleLeafModule := 15000 (* Definition of the dwModuleType for the module *)
)UDINT;
END_TYPE

// LMC_PacDrive/Application/TemplateFullProgrammingFramework/Examples/ExampleLeafModule/ST_ExampleLeafModuleInterface
TYPE ST_ExampleLeafModuleInterface :
STRUCT
	i_ifDrive						: SystemConfigurationItf.IF_Drive;
	i_lrPosMin						: LREAL;
	i_lrPosMax						: LREAL;
	i_xInitHoming					: BOOL;
	i_xEnableRandomExceptionTrigger	: BOOL;
	
	q_xValue						: BOOL := FALSE;
	q_etState						: ET_ExampleLeafModuleState := ET_ExampleLeafModuleState.Disabled;
END_STRUCT
END_TYPE

// LMC_PacDrive/Application/TemplateFullProgrammingFramework/EquipmentModules/MulticarrierModule/Multicarrier Stations/ST_StationParameter
TYPE ST_StationParameter :
STRUCT
	ifTargetStation					: MCRS.IF_CoreStation;
	
	//-- motion parameter 
	lrMaxVelocity					: LREAL;
	lrMaxAcceleration				: LREAL;
	lrMaxDeceleration				: LREAL;
	lrMaxJerk						: LREAL;
	
	//--- station parameter
	udiStationId					: UDINT;	
	lrProcessPos					: LREAL;
	lrProcessGap					: LREAL;
	lrWaitStationPosition			: LREAL;
	lrQueueGapAtWaitPos				: LREAL;
	
	//--- timer for simulation 
	diActualTime					: DINT;
	diWaitingTime					: DINT;
	xStartTimer						: BOOL;
	
	//--- miscellaneous
	xInitParameter					: BOOL;
	xTrigger						: BOOL;
	xApplicationLoggerEntriesActive	: BOOL;

	
END_STRUCT
END_TYPE

// LMC_PacDrive/Application/TemplateFullProgrammingFramework/EquipmentModules/MulticarrierModule/Multicarrier Stations/Test Multicarrier/ST_CarrierMotionData
TYPE ST_CarrierMotionData :
STRUCT
	lrVelocity			: LREAL;
	lrAcceleration		: LREAL;
	lrDeceleration		: LREAL;
	lrJerk				: LREAL;
	lrEndtarget			: LREAL;
	etPosMode			: MCR.ET_PosMode;
	lrTargetGap			: LREAL;
	
END_STRUCT
END_TYPE

// LMC_PacDrive/Application/TemplateFullProgrammingFramework/EquipmentModules/MulticarrierModule/Multicarrier Stations/Test Multicarrier/ST_EmulationTestStations
TYPE ST_EmulationTestStations :
STRUCT
	sName 				: STRING;
	lrWaitPosition 		: LREAL;
	lrProcessPosition 	: LREAL;	
	etStationColor      : DTC.ET_EmulationColors;
	udiStationId		: UDINT;
END_STRUCT
END_TYPE

// LMC_PacDrive/Application/TemplateFullProgrammingFramework/EquipmentModules/MulticarrierModule/Multicarrier Stations/AutomaticMode/Base Station/ET_ResultSource
{attribute 'qualified_only'}
{attribute 'strict'}
TYPE ET_ResultSource :
(
	Multicarrier		:= 21,
	MulticarrierStation := 22,
	UserStation			:= 6
)UDINT;
END_TYPE

// LMC_PacDrive/Application/TemplateFullProgrammingFramework/EquipmentModules/MulticarrierModule/Multicarrier Stations/AutomaticMode/Base Station/ET_ResultStation
{attribute 'qualified_only'}
{attribute 'to_string'}


TYPE ET_ResultStation :
(
	OK,							
	InvalidInput,
	WarmstartNotPossible				
	
)UINT;
END_TYPE

// LMC_PacDrive/Application/TemplateFullProgrammingFramework/EquipmentModules/MulticarrierModule/Multicarrier Stations/AutomaticMode/Base Station/ET_StationType
{attribute 'qualified_only'}
{attribute 'strict'}
TYPE ET_StationType :
(
	Load,Fill,Unload,Close,Blue, Red, Yellow,Sync, Wait
);
END_TYPE

// LMC_PacDrive/Application/MulticarrierConfiguration/GVL_MulticarrierConfiguration
{attribute 'qualified_only' := ''}
// generated content
// if modified, data can be read back to Multicarrier Configuration editor
// but will be overwritten on next update
VAR_GLOBAL CONSTANT

	/// Track configuration
	Gc_udiNumberOfTracks: UDINT := 1;
	Gc_udiMaxNumberOfSegments: UDINT := 20;
	Gc_udiMaxNumberOfStations: UDINT := 0;
	Gc_astTracks: ARRAY [1..Gc_udiNumberOfTracks] OF ST_Track := [
		(xIsClosed := TRUE, lrLength := 5208, xDirection := TRUE, lrLogicalStartOffset := 0, udiNumberOfSegments := 20, 
		 astSegments := [
			(diSegmentTypesIndex := 1),
			(diSegmentTypesIndex := 1),
			(diSegmentTypesIndex := 1),
			(diSegmentTypesIndex := 1),
			(diSegmentTypesIndex := 1),
			(diSegmentTypesIndex := 1),
			(diSegmentTypesIndex := 2),
			(diSegmentTypesIndex := 2),
			(diSegmentTypesIndex := 2),
			(diSegmentTypesIndex := 2),
			(diSegmentTypesIndex := 1),
			(diSegmentTypesIndex := 1),
			(diSegmentTypesIndex := 1),
			(diSegmentTypesIndex := 1),
			(diSegmentTypesIndex := 1),
			(diSegmentTypesIndex := 1),
			(diSegmentTypesIndex := 2),
			(diSegmentTypesIndex := 2),
			(diSegmentTypesIndex := 2),
			(diSegmentTypesIndex := 2)], 
		 udiNumberOfStations := 0, 
		 astStations := [])];
	Gc_udiNumberOfSegmentTypes: UDINT := 2;
	Gc_astSegmentTypes: ARRAY [1..Gc_udiNumberOfSegmentTypes] OF ST_SegmentType := [
		(lrRailLength := 300.4, xIsCurved := FALSE, lrAngle := 0, diAngleFractionNumerator := 0, udiAngleFractionDenominator := 1),
		(lrRailLength := 200.4, xIsCurved := TRUE, lrAngle := 45, diAngleFractionNumerator := 1, udiAngleFractionDenominator := 8)];

	/// Carrier configuration
	Gc_udiNumberOfCarrierCompounds: UDINT := 0;
	Gc_astCarrierCompounds: ARRAY [1..Gc_udiNumberOfCarrierCompounds] OF ST_CarrierCompound := [];
	Gc_udiNumberOfCarriers: UDINT := 20;
	Gc_astCarriers: ARRAY [1..Gc_udiNumberOfCarriers] OF ST_Carrier := [
		(diCarrierCompoundsIndex := 0),
		(diCarrierCompoundsIndex := 0),
		(diCarrierCompoundsIndex := 0),
		(diCarrierCompoundsIndex := 0),
		(diCarrierCompoundsIndex := 0),
		(diCarrierCompoundsIndex := 0),
		(diCarrierCompoundsIndex := 0),
		(diCarrierCompoundsIndex := 0),
		(diCarrierCompoundsIndex := 0),
		(diCarrierCompoundsIndex := 0),
		(diCarrierCompoundsIndex := 0),
		(diCarrierCompoundsIndex := 0),
		(diCarrierCompoundsIndex := 0),
		(diCarrierCompoundsIndex := 0),
		(diCarrierCompoundsIndex := 0),
		(diCarrierCompoundsIndex := 0),
		(diCarrierCompoundsIndex := 0),
		(diCarrierCompoundsIndex := 0),
		(diCarrierCompoundsIndex := 0),
		(diCarrierCompoundsIndex := 0)];

	/// Tool configuration
	Gc_udiNumberOfToolTypes: UDINT := 0;
	Gc_astToolTypes: ARRAY [1..Gc_udiNumberOfToolTypes] OF ST_ToolType := [];

	/// Tool Parts configuration
	Gc_udiNumberOfToolPartTypes: UDINT := 0;
	Gc_astToolPartTypes: ARRAY [1..Gc_udiNumberOfToolPartTypes] OF ST_PartType := [];
	Gc_udiNumberOfToolParts: UDINT := 0;
	Gc_astToolParts: ARRAY [1..Gc_udiNumberOfToolParts] OF ST_Part := [];

	/// Product configuration
	Gc_udiNumberOfProductTypes: UDINT := 0;
	Gc_astProductTypes: ARRAY [1..Gc_udiNumberOfProductTypes] OF ST_ProductType := [];
END_VAR

// LMC_PacDrive/Application/MulticarrierEmulation/GVL_MulticarrierEmulation
{attribute 'qualified_only'}
VAR_GLOBAL
	G_astPositionXYZ_Tracks : ARRAY [1..GVL_MulticarrierConfiguration.Gc_udiNumberOfTracks] OF SE_MATH.ST_Vector3D;
	G_astOrientationrXrYrZ_Tracks : ARRAY [1..GVL_MulticarrierConfiguration.Gc_udiNumberOfTracks] OF SE_MATH.ST_Vector3D;
	G_aetTrackColor : ARRAY [1..GVL_MulticarrierConfiguration.Gc_udiNumberOfTracks] OF DTC.ET_EmulationColors;

	G_audiCarriersTrackID : ARRAY [1..GVL_MulticarrierConfiguration.Gc_udiNumberOfCarriers] OF UDINT;
	G_aetCarrierColor : ARRAY [1..GVL_MulticarrierConfiguration.Gc_udiNumberOfCarriers] OF DTC.ET_EmulationColors;

	G_asStationFamily : ARRAY [1..DTC.GPL.Gc_udiMaxNumberOfStations] OF STRING(80);
	G_aetStationColor : ARRAY [1..DTC.GPL.Gc_udiMaxNumberOfStations] OF DTC.ET_EmulationColors;
	G_audiStationId : ARRAY [1..DTC.GPL.Gc_udiMaxNumberOfStations] OF UDINT;

	G_asToolFamily : ARRAY [1..GVL_MulticarrierConfiguration.Gc_udiNumberOfCarriers] OF STRING(80);
	G_astToolDimensions : ARRAY [1..GVL_MulticarrierConfiguration.Gc_udiNumberOfCarriers] OF MCR.ST_Dimensions;
	G_astToolOffsets : ARRAY [1..GVL_MulticarrierConfiguration.Gc_udiNumberOfCarriers] OF SE_MATH.ST_Vector3D;
	G_aetToolColor : ARRAY [1..GVL_MulticarrierConfiguration.Gc_udiNumberOfCarriers] OF DTC.ET_EmulationColors;

	G_asProductFamily : ARRAY [1..GVL_MulticarrierConfiguration.Gc_udiNumberOfCarriers] OF STRING(80);
	G_astProductDimensions : ARRAY [1..GVL_MulticarrierConfiguration.Gc_udiNumberOfCarriers] OF MCR.ST_Dimensions;
	G_astProductOffsets : ARRAY [1..GVL_MulticarrierConfiguration.Gc_udiNumberOfCarriers] OF SE_MATH.ST_Vector3D;
	G_aetProductColor : ARRAY [1..GVL_MulticarrierConfiguration.Gc_udiNumberOfCarriers] OF DTC.ET_EmulationColors;

	G_axCarrierCrash : ARRAY [1..GVL_MulticarrierConfiguration.Gc_udiNumberOfCarriers] OF BOOL;

	G_stDefaultDimensions : MCR.ST_Dimensions := (lrLength := 0, lrWidth := 0, lrHeight := 0);
	G_stDefaultVector3D : SE_MATH.ST_Vector3D := (lrX := 0, lrY := 0, lrZ := 0);
	G_stDefaultTrackPosition : SE_MATH.ST_Vector3D := (lrX := 0, lrY := 0, lrZ := 1000);
END_VAR

// LMC_PacDrive/Application/TemplateFullProgrammingFramework/GlobalVariables/Diagnostics
VAR_GLOBAL
	G_stDiagnosticsToApplicationMarkerarea AT %MB0 : TPL.ST_DiagnosticsToApplicationMarkerArea;
END_VAR

// LMC_PacDrive/Application/TemplateFullProgrammingFramework/GlobalVariables/ExceptionHandling
VAR_GLOBAL
	G_stExceptionList		: TPL.ST_ExceptionList;
END_VAR

// LMC_PacDrive/Application/TemplateFullProgrammingFramework/GlobalVariables/GVL_Project
{attribute 'qualified_only'}
VAR_GLOBAL CONSTANT
	Gc_xVirtualMulticarrier				: BOOL := TRUE;
	Gc_xEnableCrashPrevention			: BOOL := TRUE;
	Gc_xTrackCalibrationOfMulticarrier	: BOOL := FALSE;
END_VAR

VAR_GLOBAL
	G_udiUsedNumberOfCarriers			: UDINT; //no initialisation needed -> is set in SR_MainMachine.Start_Action 
	G_xEnableAplEntriesViaStation		: BOOL;
	G_lrCrashDistance					: LREAL := 5; // is the distance of the front offset of carrier and the rear offset of the next carrier
	
	// /!\ Variables for Emulation
	G_udiMaxNumberOfStations 			: UDINT := 6;	
	G_astEmulationStations 				: ARRAY [1..6] OF DTC.ST_StationConfig;	
	
END_VAR

// LMC_PacDrive/Application/TemplateFullProgrammingFramework/GlobalVariables/HardwareInOuts
VAR_GLOBAL
	G_xMainsContactorOut 		(*-AT %QX0.0-*)	: BOOL;

	G_xEmergencyIn  			(*-AT %IX0.0-*)	: BOOL;
	G_xMainsContactorIn 		(*-AT %IX0.1-*)	: BOOL;
END_VAR

// LMC_PacDrive/Application/TemplateFullProgrammingFramework/GlobalVariables/InputVariablesEpas
VAR_GLOBAL
	G_xStartEpas				: BOOL;
	G_xStopEpas					: BOOL;
	G_xPrepareEpas				: BOOL;
	G_xAutoEpas					: BOOL;
	G_xHoldEpas					: BOOL;
	G_xAbortEpas				: BOOL;
	G_xProductsOkEpas			: BOOL;
	G_xPowerOnEpas				: BOOL;
	G_xPowerOffEpas				: BOOL;
	G_xManualEpas				: BOOL;
	G_xJogMachineEpas			: BOOL;
	G_xDiagQuitEpas				: BOOL;
	G_xEmergencyEpas			: BOOL := TRUE;
	G_xJogForwEpas				: BOOL;
	G_xJogBackEpas				: BOOL;
	G_xBrakeReleaseEpas			: BOOL;
	G_xTestMulticarrierEpas		: BOOL;
	G_xTrackCalibrationEpas		: BOOL;
	
	G_udiManualModuleSelect		: UDINT;
//	G_udiManualElementSelect	: UDINT;

	G_xDoEnableVis				: BOOL := FALSE;

	G_xDoTestMulticarrier		: BOOL;
	G_xDoPrepare 				: BOOL;
	G_xDoAuto	 				: BOOL;
	G_xDoManual 				: BOOL;
	G_xDoJogMachine 			: BOOL;
	G_xDoBrakeRelease			: BOOL;
	G_xDoTrackCalibration		: BOOL;
	
	G_xTestMulticarrierActive	: BOOL;
	G_xPrepareActive 			: BOOL;
	G_xAutoActive	 			: BOOL;
	G_xManualActive 			: BOOL;
	G_xJogMachineActive 		: BOOL;
	G_xBrakeReleaseActive		: BOOL;
	G_xTrackCalibrationActive	: BOOL;
	
	G_xStartDone				: BOOL;
END_VAR

// LMC_PacDrive/Application/TemplateFullProgrammingFramework/GlobalVariables/InputVariablesExt
VAR_GLOBAL
	G_xStartExt			: BOOL;
	G_xStopExt			: BOOL;
	G_xPrepareExt		: BOOL;
	G_xAutoExt			: BOOL;
	G_xHoldExt			: BOOL;
	G_xAbortExt			: BOOL;
	G_xProductsOkExt	: BOOL;
	G_xPowerOnExt		: BOOL;
	G_xPowerOffExt		: BOOL;
	G_xManualExt		: BOOL;
	G_xJogMachineExt	: BOOL;
	G_xDiagQuitExt		: BOOL;
	G_xJogForwExt		: BOOL;
	G_xJogBackExt		: BOOL;
	G_xBrakeReleaseExt	: BOOL;
	G_xTestMulticarrierExt	: BOOL;
	G_xTrackCalibrationExt	: BOOL;
END_VAR

// LMC_PacDrive/Application/TemplateFullProgrammingFramework/GlobalVariables/IntelligentLineShaft
VAR_GLOBAL
	G_stIlsData : PDL.ST_IlsData;
END_VAR

// LMC_PacDrive/Application/TemplateFullProgrammingFramework/GlobalVariables/Logging
VAR_GLOBAL
	G_stLogDataList			: TPL.ST_LogDataList;			(* Global log data list *)
	G_stLogDataListAscii	: TPL.ST_LogDataListAscii;		(* Temp.list for save in XML format *)
	G_stLoggerInterface		: TPL.ST_LoggerInterface;		(* Interface between logger and main machine *)
END_VAR

// LMC_PacDrive/Application/TemplateFullProgrammingFramework/GlobalVariables/RestoreAxisPosition
VAR_GLOBAL PERSISTENT RETAIN
	Grp_stRestorePositionAxis1	: PDL.ST_AxisRestorePosition;
	Grp_stRestorePositionAxis2	: PDL.ST_AxisRestorePosition;
	Grp_stRestorePositionAxis3	: PDL.ST_AxisRestorePosition;
	Grp_stRestorePositionAxis4	: PDL.ST_AxisRestorePosition;
END_VAR

// LMC_PacDrive/Application/MulticarrierEmulation/SR_EmulationInterface
// generated content, do not modify
PROGRAM SR_EmulationInterface
VAR
	xInitMulticarrierEmulationDone: BOOL := FALSE;
	udiLoop: UDINT;
	udiLoopTrack: UDINT;
	udiIndex: UDINT;
END_VAR

// generated content, do not modify
//--------------------------------------------------------------------------------------------------------------------------------
//--- Initialize
//--------------------------------------------------------------------------------------------------------------------------------
	IF NOT xInitMulticarrierEmulationDone THEN
		Init_MulticarrierEmulation();
	END_IF
	udiLoopTrack := 1;
	udiIndex := 0;

//--------------------------------------------------------------------------------------------------------------------------------
//--- Multi carrier
//--------------------------------------------------------------------------------------------------------------------------------
	//--- Track 1
		DTC.GVL_OpcUaMulticarrier.G_stMCR.astTracks[1].sCategory := 'LXMMC12';
		DTC.GVL_OpcUaMulticarrier.G_stMCR.astTracks[1].sName := 'MC_Track_1';
		DTC.GVL_OpcUaMulticarrier.G_stMCR.astTracks[1].udiColor := GVL_MulticarrierEmulation.G_aetTrackColor[1];
		DTC.GVL_OpcUaMulticarrier.G_stMCR.astTracks[1].stPosition := GVL_MulticarrierEmulation.G_astPositionXYZ_Tracks[1];
		DTC.GVL_OpcUaMulticarrier.G_stMCR.astTracks[1].stOrientation := GVL_MulticarrierEmulation.G_astOrientationrXrYrZ_Tracks[1];
		DTC.GVL_OpcUaMulticarrier.G_stMCR.astTracks[1].udiTrackID := 1;
		DTC.GVL_OpcUaMulticarrier.G_stMCR.astTracks[1].udiUnivocalId := DTC.ET_EntityOffset.Track + DTC.GVL_OpcUaMulticarrier.G_stMCR.astTracks[1].udiTrackID;
		DTC.GVL_OpcUaMulticarrier.G_stMCR.astTracks[1].xDirection := GVL_MulticarrierConfiguration.Gc_astTracks[1].xDirection;
		DTC.GVL_OpcUaMulticarrier.G_stMCR.astTracks[1].lrLogicalStartOffset := GVL_MulticarrierConfiguration.Gc_astTracks[1].lrLogicalStartOffset;

		FOR udiLoop := 1 TO MIN(GVL_Project.G_udiMaxNumberOfStations, DTC.GPL.Gc_udiMaxNumberOfStations) DO //MIN(GVL_MulticarrierConfiguration.Gc_udiMaxNumberOfStations, DTC.GPL.Gc_udiMaxNumberOfStations) DO
			udiIndex := udiIndex + 1;
			IF udiIndex > MIN(GVL_Project.G_udiMaxNumberOfStations, DTC.GPL.Gc_udiMaxNumberOfStations) THEN //GVL_MulticarrierConfiguration.Gc_astTracks[udiLoopTrack].udiNumberOfStations THEN
				udiIndex := 1;
				udiLoopTrack := udiLoopTrack + 1;
				IF udiLoopTrack > GVL_MulticarrierConfiguration.Gc_udiNumberOfTracks THEN
					EXIT;
				END_IF
			END_IF
			IF udiLoop <= DTC.GPL.Gc_udiMaxNumberOfStations THEN
				DTC.GVL_OpcUaMulticarrier.G_stMCR.astStations[udiLoop].sCategory := GVL_MulticarrierEmulation.G_asStationFamily[udiLoop];
				DTC.GVL_OpcUaMulticarrier.G_stMCR.astStations[udiLoop].udiTrackID := udiLoopTrack;
				DTC.GVL_OpcUaMulticarrier.G_stMCR.astStations[udiLoop].sTextLabel := GVL_Project.G_astEmulationStations[udiLoop].sTextLabel; //GVL_MulticarrierConfiguration.Gc_astTracks[udiLoopTrack].astStations[udiIndex].sTextLabel;
				DTC.GVL_OpcUaMulticarrier.G_stMCR.astStations[udiLoop].lrWaitPosition := GVL_Project.G_astEmulationStations[udiLoop].lrWaitPosition; //GVL_MulticarrierConfiguration.Gc_astTracks[udiLoopTrack].astStations[udiIndex].lrWaitPosition;
				DTC.GVL_OpcUaMulticarrier.G_stMCR.astStations[udiLoop].lrProcessPosition := GVL_Project.G_astEmulationStations[udiLoop].lrProcessPosition; //GVL_MulticarrierConfiguration.Gc_astTracks[udiLoopTrack].astStations[udiIndex].lrProcessPosition;
				DTC.GVL_OpcUaMulticarrier.G_stMCR.astStations[udiLoop].udiStationId := GVL_Project.G_astEmulationStations[udiLoop].udiStationId;
				DTC.GVL_OpcUaMulticarrier.G_stMCR.astStations[udiLoop].udiColor := GVL_Project.G_astEmulationStations[udiLoop].udiColor;
			END_IF
		END_FOR

	//--- Carrier Pool
		FOR udiLoop := 1 TO MIN(GVL_MulticarrierConfiguration.Gc_udiNumberOfCarriers,  MCR.GPL.Gc_udiMaxNumberOfCarriers) DO
	//--- Carrier udiLoop
			DTC.GVL_OpcUaMulticarrier.G_stMCR.astCarriers[udiLoop].sCategory := 'LXMMC12Carrier';
			DTC.GVL_OpcUaMulticarrier.G_stMCR.astCarriers[udiLoop].udiCarrierID := udiLoop;
			DTC.GVL_OpcUaMulticarrier.G_stMCR.astCarriers[udiLoop].udiUnivocalId := DTC.ET_EntityOffset.Carrier + DTC.GVL_OpcUaMulticarrier.G_stMCR.astCarriers[udiLoop].udiCarrierID;
			DTC.GVL_OpcUaMulticarrier.G_stMCR.astCarriers[udiLoop].udiColor := GVL_MulticarrierEmulation.G_aetCarrierColor[udiLoop];
			DTC.GVL_OpcUaMulticarrier.G_stMCR.astCarriers[udiLoop].udiTrackID := GVL_MulticarrierEmulation.G_audiCarriersTrackID[udiLoop];
			DTC.GVL_OpcUaMulticarrier.G_stMCR.astCarriers[udiLoop].stToolConfig.sCategory := GVL_MulticarrierEmulation.G_asToolFamily[udiLoop];
			DTC.GVL_OpcUaMulticarrier.G_stMCR.astCarriers[udiLoop].stToolConfig.stToolDimensions := GVL_MulticarrierEmulation.G_astToolDimensions[udiLoop];
			DTC.GVL_OpcUaMulticarrier.G_stMCR.astCarriers[udiLoop].stToolConfig.stToolOffset := GVL_MulticarrierEmulation.G_astToolOffsets[udiLoop];
			DTC.GVL_OpcUaMulticarrier.G_stMCR.astCarriers[udiLoop].stToolConfig.udiColor := GVL_MulticarrierEmulation.G_aetToolColor[udiLoop];
			DTC.GVL_OpcUaMulticarrier.G_stMCR.astCarriers[udiLoop].stProductConfig.sCategory := GVL_MulticarrierEmulation.G_asProductFamily[udiLoop];
			DTC.GVL_OpcUaMulticarrier.G_stMCR.astCarriers[udiLoop].stProductConfig.stProductDimensions := GVL_MulticarrierEmulation.G_astProductDimensions[udiLoop];
			DTC.GVL_OpcUaMulticarrier.G_stMCR.astCarriers[udiLoop].stProductConfig.stProductOffset := GVL_MulticarrierEmulation.G_astProductOffsets[udiLoop];
			DTC.GVL_OpcUaMulticarrier.G_stMCR.astCarriers[udiLoop].stProductConfig.udiColor := GVL_MulticarrierEmulation.G_aetProductColor[udiLoop];
			GVL_MulticarrierEmulation.G_axCarrierCrash[udiLoop] := DTC.GVL_OpcUaMulticarrier.G_stMCR.astCarriers[udiLoop].xCollisionDetection;
		END_FOR

    {IF defined (variable:MC_Carrier_1)}
		DTC.GVL_OpcUaMulticarrier.G_stMCR.astCarriers[1].lrPositionX := MC_Carrier_1.MovementData.RefPosition;
    {END_IF}
    {IF defined (variable:MC_Carrier_2)}
		DTC.GVL_OpcUaMulticarrier.G_stMCR.astCarriers[2].lrPositionX := MC_Carrier_2.MovementData.RefPosition;
    {END_IF}
    {IF defined (variable:MC_Carrier_3)}
		DTC.GVL_OpcUaMulticarrier.G_stMCR.astCarriers[3].lrPositionX := MC_Carrier_3.MovementData.RefPosition;
    {END_IF}
    {IF defined (variable:MC_Carrier_4)}
		DTC.GVL_OpcUaMulticarrier.G_stMCR.astCarriers[4].lrPositionX := MC_Carrier_4.MovementData.RefPosition;
    {END_IF}
    {IF defined (variable:MC_Carrier_5)}
		DTC.GVL_OpcUaMulticarrier.G_stMCR.astCarriers[5].lrPositionX := MC_Carrier_5.MovementData.RefPosition;
    {END_IF}
    {IF defined (variable:MC_Carrier_6)}
		DTC.GVL_OpcUaMulticarrier.G_stMCR.astCarriers[6].lrPositionX := MC_Carrier_6.MovementData.RefPosition;
    {END_IF}
    {IF defined (variable:MC_Carrier_7)}
		DTC.GVL_OpcUaMulticarrier.G_stMCR.astCarriers[7].lrPositionX := MC_Carrier_7.MovementData.RefPosition;
    {END_IF}
    {IF defined (variable:MC_Carrier_8)}
		DTC.GVL_OpcUaMulticarrier.G_stMCR.astCarriers[8].lrPositionX := MC_Carrier_8.MovementData.RefPosition;
    {END_IF}
    {IF defined (variable:MC_Carrier_9)}
		DTC.GVL_OpcUaMulticarrier.G_stMCR.astCarriers[9].lrPositionX := MC_Carrier_9.MovementData.RefPosition;
    {END_IF}
    {IF defined (variable:MC_Carrier_10)}
		DTC.GVL_OpcUaMulticarrier.G_stMCR.astCarriers[10].lrPositionX := MC_Carrier_10.MovementData.RefPosition;
    {END_IF}
    {IF defined (variable:MC_Carrier_11)}
		DTC.GVL_OpcUaMulticarrier.G_stMCR.astCarriers[11].lrPositionX := MC_Carrier_11.MovementData.RefPosition;
    {END_IF}
    {IF defined (variable:MC_Carrier_12)}
		DTC.GVL_OpcUaMulticarrier.G_stMCR.astCarriers[12].lrPositionX := MC_Carrier_12.MovementData.RefPosition;
    {END_IF}
    {IF defined (variable:MC_Carrier_13)}
		DTC.GVL_OpcUaMulticarrier.G_stMCR.astCarriers[13].lrPositionX := MC_Carrier_13.MovementData.RefPosition;
    {END_IF}
    {IF defined (variable:MC_Carrier_14)}
		DTC.GVL_OpcUaMulticarrier.G_stMCR.astCarriers[14].lrPositionX := MC_Carrier_14.MovementData.RefPosition;
    {END_IF}
    {IF defined (variable:MC_Carrier_15)}
		DTC.GVL_OpcUaMulticarrier.G_stMCR.astCarriers[15].lrPositionX := MC_Carrier_15.MovementData.RefPosition;
    {END_IF}
    {IF defined (variable:MC_Carrier_16)}
		DTC.GVL_OpcUaMulticarrier.G_stMCR.astCarriers[16].lrPositionX := MC_Carrier_16.MovementData.RefPosition;
    {END_IF}
    {IF defined (variable:MC_Carrier_17)}
		DTC.GVL_OpcUaMulticarrier.G_stMCR.astCarriers[17].lrPositionX := MC_Carrier_17.MovementData.RefPosition;
    {END_IF}
    {IF defined (variable:MC_Carrier_18)}
		DTC.GVL_OpcUaMulticarrier.G_stMCR.astCarriers[18].lrPositionX := MC_Carrier_18.MovementData.RefPosition;
    {END_IF}
    {IF defined (variable:MC_Carrier_19)}
		DTC.GVL_OpcUaMulticarrier.G_stMCR.astCarriers[19].lrPositionX := MC_Carrier_19.MovementData.RefPosition;
    {END_IF}
    {IF defined (variable:MC_Carrier_20)}
		DTC.GVL_OpcUaMulticarrier.G_stMCR.astCarriers[20].lrPositionX := MC_Carrier_20.MovementData.RefPosition;
    {END_IF}
    {IF defined (variable:MC_Carrier_21)}
		DTC.GVL_OpcUaMulticarrier.G_stMCR.astCarriers[21].lrPositionX := MC_Carrier_21.MovementData.RefPosition;
    {END_IF}
    {IF defined (variable:MC_Carrier_22)}
		DTC.GVL_OpcUaMulticarrier.G_stMCR.astCarriers[22].lrPositionX := MC_Carrier_22.MovementData.RefPosition;
    {END_IF}
    {IF defined (variable:MC_Carrier_23)}
		DTC.GVL_OpcUaMulticarrier.G_stMCR.astCarriers[23].lrPositionX := MC_Carrier_23.MovementData.RefPosition;
    {END_IF}
    {IF defined (variable:MC_Carrier_24)}
		DTC.GVL_OpcUaMulticarrier.G_stMCR.astCarriers[24].lrPositionX := MC_Carrier_24.MovementData.RefPosition;
    {END_IF}
    {IF defined (variable:MC_Carrier_25)}
		DTC.GVL_OpcUaMulticarrier.G_stMCR.astCarriers[25].lrPositionX := MC_Carrier_25.MovementData.RefPosition;
    {END_IF}
    {IF defined (variable:MC_Carrier_26)}
		DTC.GVL_OpcUaMulticarrier.G_stMCR.astCarriers[26].lrPositionX := MC_Carrier_26.MovementData.RefPosition;
    {END_IF}
    {IF defined (variable:MC_Carrier_27)}
		DTC.GVL_OpcUaMulticarrier.G_stMCR.astCarriers[27].lrPositionX := MC_Carrier_27.MovementData.RefPosition;
    {END_IF}
    {IF defined (variable:MC_Carrier_28)}
		DTC.GVL_OpcUaMulticarrier.G_stMCR.astCarriers[28].lrPositionX := MC_Carrier_28.MovementData.RefPosition;
    {END_IF}
    {IF defined (variable:MC_Carrier_29)}
		DTC.GVL_OpcUaMulticarrier.G_stMCR.astCarriers[29].lrPositionX := MC_Carrier_29.MovementData.RefPosition;
    {END_IF}
    {IF defined (variable:MC_Carrier_30)}
		DTC.GVL_OpcUaMulticarrier.G_stMCR.astCarriers[30].lrPositionX := MC_Carrier_30.MovementData.RefPosition;
    {END_IF}
    {IF defined (variable:MC_Carrier_31)}
		DTC.GVL_OpcUaMulticarrier.G_stMCR.astCarriers[31].lrPositionX := MC_Carrier_31.MovementData.RefPosition;
    {END_IF}
    {IF defined (variable:MC_Carrier_32)}
		DTC.GVL_OpcUaMulticarrier.G_stMCR.astCarriers[32].lrPositionX := MC_Carrier_32.MovementData.RefPosition;
    {END_IF}
    {IF defined (variable:MC_Carrier_33)}
		DTC.GVL_OpcUaMulticarrier.G_stMCR.astCarriers[33].lrPositionX := MC_Carrier_33.MovementData.RefPosition;
    {END_IF}
    {IF defined (variable:MC_Carrier_34)}
		DTC.GVL_OpcUaMulticarrier.G_stMCR.astCarriers[34].lrPositionX := MC_Carrier_34.MovementData.RefPosition;
    {END_IF}
    {IF defined (variable:MC_Carrier_35)}
		DTC.GVL_OpcUaMulticarrier.G_stMCR.astCarriers[35].lrPositionX := MC_Carrier_35.MovementData.RefPosition;
    {END_IF}
    {IF defined (variable:MC_Carrier_36)}
		DTC.GVL_OpcUaMulticarrier.G_stMCR.astCarriers[36].lrPositionX := MC_Carrier_36.MovementData.RefPosition;
    {END_IF}
    {IF defined (variable:MC_Carrier_37)}
		DTC.GVL_OpcUaMulticarrier.G_stMCR.astCarriers[37].lrPositionX := MC_Carrier_37.MovementData.RefPosition;
    {END_IF}
    {IF defined (variable:MC_Carrier_38)}
		DTC.GVL_OpcUaMulticarrier.G_stMCR.astCarriers[38].lrPositionX := MC_Carrier_38.MovementData.RefPosition;
    {END_IF}
    {IF defined (variable:MC_Carrier_39)}
		DTC.GVL_OpcUaMulticarrier.G_stMCR.astCarriers[39].lrPositionX := MC_Carrier_39.MovementData.RefPosition;
    {END_IF}
    {IF defined (variable:MC_Carrier_40)}
		DTC.GVL_OpcUaMulticarrier.G_stMCR.astCarriers[40].lrPositionX := MC_Carrier_40.MovementData.RefPosition;
    {END_IF}
    {IF defined (variable:MC_Carrier_41)}
		DTC.GVL_OpcUaMulticarrier.G_stMCR.astCarriers[41].lrPositionX := MC_Carrier_41.MovementData.RefPosition;
    {END_IF}
    {IF defined (variable:MC_Carrier_42)}
		DTC.GVL_OpcUaMulticarrier.G_stMCR.astCarriers[42].lrPositionX := MC_Carrier_42.MovementData.RefPosition;
    {END_IF}
    {IF defined (variable:MC_Carrier_43)}
		DTC.GVL_OpcUaMulticarrier.G_stMCR.astCarriers[43].lrPositionX := MC_Carrier_43.MovementData.RefPosition;
    {END_IF}
    {IF defined (variable:MC_Carrier_44)}
		DTC.GVL_OpcUaMulticarrier.G_stMCR.astCarriers[44].lrPositionX := MC_Carrier_44.MovementData.RefPosition;
    {END_IF}
    {IF defined (variable:MC_Carrier_45)}
		DTC.GVL_OpcUaMulticarrier.G_stMCR.astCarriers[45].lrPositionX := MC_Carrier_45.MovementData.RefPosition;
    {END_IF}
    {IF defined (variable:MC_Carrier_46)}
		DTC.GVL_OpcUaMulticarrier.G_stMCR.astCarriers[46].lrPositionX := MC_Carrier_46.MovementData.RefPosition;
    {END_IF}
    {IF defined (variable:MC_Carrier_47)}
		DTC.GVL_OpcUaMulticarrier.G_stMCR.astCarriers[47].lrPositionX := MC_Carrier_47.MovementData.RefPosition;
    {END_IF}
    {IF defined (variable:MC_Carrier_48)}
		DTC.GVL_OpcUaMulticarrier.G_stMCR.astCarriers[48].lrPositionX := MC_Carrier_48.MovementData.RefPosition;
    {END_IF}
    {IF defined (variable:MC_Carrier_49)}
		DTC.GVL_OpcUaMulticarrier.G_stMCR.astCarriers[49].lrPositionX := MC_Carrier_49.MovementData.RefPosition;
    {END_IF}
    {IF defined (variable:MC_Carrier_50)}
		DTC.GVL_OpcUaMulticarrier.G_stMCR.astCarriers[50].lrPositionX := MC_Carrier_50.MovementData.RefPosition;
    {END_IF}
    {IF defined (variable:MC_Carrier_51)}
		DTC.GVL_OpcUaMulticarrier.G_stMCR.astCarriers[51].lrPositionX := MC_Carrier_51.MovementData.RefPosition;
    {END_IF}
    {IF defined (variable:MC_Carrier_52)}
		DTC.GVL_OpcUaMulticarrier.G_stMCR.astCarriers[52].lrPositionX := MC_Carrier_52.MovementData.RefPosition;
    {END_IF}
    {IF defined (variable:MC_Carrier_53)}
		DTC.GVL_OpcUaMulticarrier.G_stMCR.astCarriers[53].lrPositionX := MC_Carrier_53.MovementData.RefPosition;
    {END_IF}
    {IF defined (variable:MC_Carrier_54)}
		DTC.GVL_OpcUaMulticarrier.G_stMCR.astCarriers[54].lrPositionX := MC_Carrier_54.MovementData.RefPosition;
    {END_IF}
    {IF defined (variable:MC_Carrier_55)}
		DTC.GVL_OpcUaMulticarrier.G_stMCR.astCarriers[55].lrPositionX := MC_Carrier_55.MovementData.RefPosition;
    {END_IF}
    {IF defined (variable:MC_Carrier_56)}
		DTC.GVL_OpcUaMulticarrier.G_stMCR.astCarriers[56].lrPositionX := MC_Carrier_56.MovementData.RefPosition;
    {END_IF}
    {IF defined (variable:MC_Carrier_57)}
		DTC.GVL_OpcUaMulticarrier.G_stMCR.astCarriers[57].lrPositionX := MC_Carrier_57.MovementData.RefPosition;
    {END_IF}
    {IF defined (variable:MC_Carrier_58)}
		DTC.GVL_OpcUaMulticarrier.G_stMCR.astCarriers[58].lrPositionX := MC_Carrier_58.MovementData.RefPosition;
    {END_IF}
    {IF defined (variable:MC_Carrier_59)}
		DTC.GVL_OpcUaMulticarrier.G_stMCR.astCarriers[59].lrPositionX := MC_Carrier_59.MovementData.RefPosition;
    {END_IF}
    {IF defined (variable:MC_Carrier_60)}
		DTC.GVL_OpcUaMulticarrier.G_stMCR.astCarriers[60].lrPositionX := MC_Carrier_60.MovementData.RefPosition;
    {END_IF}
    {IF defined (variable:MC_Carrier_61)}
		DTC.GVL_OpcUaMulticarrier.G_stMCR.astCarriers[61].lrPositionX := MC_Carrier_61.MovementData.RefPosition;
    {END_IF}
    {IF defined (variable:MC_Carrier_62)}
		DTC.GVL_OpcUaMulticarrier.G_stMCR.astCarriers[62].lrPositionX := MC_Carrier_62.MovementData.RefPosition;
    {END_IF}
    {IF defined (variable:MC_Carrier_63)}
		DTC.GVL_OpcUaMulticarrier.G_stMCR.astCarriers[63].lrPositionX := MC_Carrier_63.MovementData.RefPosition;
    {END_IF}
    {IF defined (variable:MC_Carrier_64)}
		DTC.GVL_OpcUaMulticarrier.G_stMCR.astCarriers[64].lrPositionX := MC_Carrier_64.MovementData.RefPosition;
    {END_IF}
    {IF defined (variable:MC_Carrier_65)}
		DTC.GVL_OpcUaMulticarrier.G_stMCR.astCarriers[65].lrPositionX := MC_Carrier_65.MovementData.RefPosition;
    {END_IF}
    {IF defined (variable:MC_Carrier_66)}
		DTC.GVL_OpcUaMulticarrier.G_stMCR.astCarriers[66].lrPositionX := MC_Carrier_66.MovementData.RefPosition;
    {END_IF}
    {IF defined (variable:MC_Carrier_67)}
		DTC.GVL_OpcUaMulticarrier.G_stMCR.astCarriers[67].lrPositionX := MC_Carrier_67.MovementData.RefPosition;
    {END_IF}
    {IF defined (variable:MC_Carrier_68)}
		DTC.GVL_OpcUaMulticarrier.G_stMCR.astCarriers[68].lrPositionX := MC_Carrier_68.MovementData.RefPosition;
    {END_IF}
    {IF defined (variable:MC_Carrier_69)}
		DTC.GVL_OpcUaMulticarrier.G_stMCR.astCarriers[69].lrPositionX := MC_Carrier_69.MovementData.RefPosition;
    {END_IF}
    {IF defined (variable:MC_Carrier_70)}
		DTC.GVL_OpcUaMulticarrier.G_stMCR.astCarriers[70].lrPositionX := MC_Carrier_70.MovementData.RefPosition;
    {END_IF}

METHOD Init_MulticarrierEmulation
VAR
END_VAR
// generated content, do not modify
//--- Tracks
	//--- Set Position
		FOR udiLoop := 1 TO GVL_MulticarrierConfiguration.Gc_udiNumberOfTracks DO
			GVL_MulticarrierEmulation.G_astPositionXYZ_Tracks[udiLoop]:= GVL_MulticarrierEmulation.G_stDefaultTrackPosition;
		END_FOR

	//--- Set Orientation
		FOR udiLoop := 1 TO GVL_MulticarrierConfiguration.Gc_udiNumberOfTracks DO
			GVL_MulticarrierEmulation.G_astOrientationrXrYrZ_Tracks[udiLoop]:= GVL_MulticarrierEmulation.G_stDefaultVector3D;
		END_FOR

	//--- Set Color
		FOR udiLoop := 1 TO GVL_MulticarrierConfiguration.Gc_udiNumberOfTracks DO
			GVL_MulticarrierEmulation.G_aetTrackColor[udiLoop]:= DTC.ET_EmulationColors.None;
		END_FOR

//--- Stations
	//--- Set Family
		FOR udiLoop := 1 TO DTC.GPL.Gc_udiMaxNumberOfStations DO
			GVL_MulticarrierEmulation.G_asStationFamily[udiLoop]:= 'StandardStation';
		END_FOR

	//--- Set Color
		FOR udiLoop := 1 TO DTC.GPL.Gc_udiMaxNumberOfStations DO
			GVL_MulticarrierEmulation.G_aetStationColor[udiLoop]:= DTC.ET_EmulationColors.Black;
		END_FOR

	//--- Set Station Id
		FOR udiLoop := 1 TO DTC.GPL.Gc_udiMaxNumberOfStations DO
			GVL_MulticarrierEmulation.G_audiStationId[udiLoop]:= udiLoop;
		END_FOR

//--- Carriers
	//--- Set Track-ID
		FOR udiLoop := 1 TO GVL_MulticarrierConfiguration.Gc_udiNumberOfCarriers DO
			GVL_MulticarrierEmulation.G_audiCarriersTrackID[udiLoop]:= 1;
		END_FOR

	//--- Set Color
		FOR udiLoop := 1 TO GVL_MulticarrierConfiguration.Gc_udiNumberOfCarriers DO
			IF udiLoop = 1 THEN
				GVL_MulticarrierEmulation.G_aetCarrierColor[udiLoop] := DTC.ET_EmulationColors.LimeGreen;
			ELSE
				GVL_MulticarrierEmulation.G_aetCarrierColor[udiLoop] := DTC.ET_EmulationColors.None;
			END_IF
		END_FOR

	//--- Set Tool Family
		FOR udiLoop := 1 TO GVL_MulticarrierConfiguration.Gc_udiNumberOfCarriers DO
			GVL_MulticarrierEmulation.G_asToolFamily[udiLoop]:= 'StandardTool';
		END_FOR

	//--- Set Tool Dimensions
		FOR udiLoop := 1 TO GVL_MulticarrierConfiguration.Gc_udiNumberOfCarriers DO
			GVL_MulticarrierEmulation.G_astToolDimensions[udiLoop]:= GVL_MulticarrierEmulation.G_stDefaultDimensions;
		END_FOR

	//--- Set Tool Offset
		FOR udiLoop := 1 TO GVL_MulticarrierConfiguration.Gc_udiNumberOfCarriers DO
			GVL_MulticarrierEmulation.G_astToolOffsets[udiLoop]:= GVL_MulticarrierEmulation.G_stDefaultVector3D;
		END_FOR

	//--- Set Tool Color
		FOR udiLoop := 1 TO GVL_MulticarrierConfiguration.Gc_udiNumberOfCarriers DO
			GVL_MulticarrierEmulation.G_aetToolColor[udiLoop]:= DTC.ET_EmulationColors.DarkSlateGray;
		END_FOR

	//--- Set Product Family
		FOR udiLoop := 1 TO GVL_MulticarrierConfiguration.Gc_udiNumberOfCarriers DO
			GVL_MulticarrierEmulation.G_asProductFamily[udiLoop]:= 'StandardProduct';
		END_FOR

	//--- Set Product Dimensions
		FOR udiLoop := 1 TO GVL_MulticarrierConfiguration.Gc_udiNumberOfCarriers DO
			GVL_MulticarrierEmulation.G_astProductDimensions[udiLoop]:= GVL_MulticarrierEmulation.G_stDefaultDimensions;
		END_FOR

	//--- Set Product Offset
		FOR udiLoop := 1 TO GVL_MulticarrierConfiguration.Gc_udiNumberOfCarriers DO
			GVL_MulticarrierEmulation.G_astProductOffsets[udiLoop]:= GVL_MulticarrierEmulation.G_stDefaultVector3D;
		END_FOR

	//--- Set Product Color
		FOR udiLoop := 1 TO GVL_MulticarrierConfiguration.Gc_udiNumberOfCarriers DO
			GVL_MulticarrierEmulation.G_aetProductColor[udiLoop]:= DTC.ET_EmulationColors.Transparent;
		END_FOR

xInitMulticarrierEmulationDone := TRUE;
END_METHOD

END_PROGRAM

// LMC_PacDrive/Application/TemplateFullProgrammingFramework/TaskCalls/SR_OpcUa
PROGRAM SR_OpcUa
VAR
	byState						: BYTE := 0;
	///Control OPC UA 
	diResultStartOpcUa			: DINT := 0;
	diResultStopOpcUa			: DINT := 0;
	xStartUaServer				: BOOL := TRUE;
	stOpcUaServerConfig			: SystemInterface.ST_ExternalOpcUaServerConfig;
	xCallOnceWhenStopServer		: BOOL := TRUE;
	///Fast Item access on/off -> if 'off' no Parameter access via OPC UA supported
	xActivateFastAcc			: BOOL := TRUE;
	diResultOpcUaSetAccessType	: DINT;
	///Control Cycle Time check
	diAddOverrunTimeSum			: DINT := 0;
	diAddWDogTimeSum			: DINT := 0;
	diOverrunTime				: DINT;
	diWDogTime					: DINT;
	diAddOverrunTime			: DINT;
	diAddWDogTime				: DINT;
	END_VAR

// opc.tcp://*enter_PLC_IP_Address*:*enter_Port_nummber*
// Port is 4840

// Reset CycleCheckTime at the beginning of next cycle whenever it was increased
IF diAddOverrunTimeSum > 0 OR diAddWDogTimeSum > 0 THEN
	SystemInterface.FC_CycleCheckTimeGet(iq_diOverrunTime := diOverrunTime, iq_diWDogFactor := diWDogTime);
	SystemInterface.FC_CycleCheckTimeSet(i_diOverrunTime := (diOverrunTime - diAddOverrunTimeSum), i_diWDogFactor := (diWDogTime - diAddWDogTimeSum));
	
	diAddOverrunTimeSum := 0;
	diAddWDogTimeSum := 0;
END_IF;


// ---------------------------- START OPC UA SERVER ----------------------------------
CASE byState OF

	0: 	// Wait until main programm is started
		IF SR_MainMachine.xInitSuccessful THEN
			// Activation/Deactivation of OPC UA fast access
			IF xActivateFastAcc THEN
				diResultOpcUaSetAccessType := Systeminterface.FC_OpcUaSetAccessType(i_etOpcUaAccessType := ET_OpcUaAccessType.MEMORYACC);
			ELSE
				diResultOpcUaSetAccessType := Systeminterface.FC_OpcUaSetAccessType(i_etOpcUaAccessType := ET_OpcUaAccessType.IECVARACC);
			END_IF
			
			byState:=	5;
		END_IF	
		
	5:	// Start Command to start OPC UA Server
		IF xStartUaServer THEN
			xCallOnceWhenStopServer := TRUE;
			SystemInterface.FC_FirewallSetActive(i_xActive := FALSE); 
			byState:=	10;
		END_IF	

	10:	// Increase CycleCheckTime for one Cycle
		diAddOverrunTime := 500 ;
		diAddWDogTime 	 := 2000;
		
		SystemInterface.FC_CycleCheckTimeGet(iq_diOverrunTime := diOverrunTime, iq_diWDogFactor := diWDogTime);
		SystemInterface.FC_CycleCheckTimeSet(i_diOverrunTime := (diOverrunTime + diAddOverrunTime), i_diWDogFactor := (diWDogTime + diAddWDogTime));
		
		diAddOverrunTimeSum := diAddOverrunTimeSum + diAddOverrunTime;
		diAddWDogTimeSum := diAddWDogTimeSum + diAddWDogTime;
		
		// Start OPC UA server 
		diResultStartOpcUa := SystemInterface.FC_OpcUaStart('Schneider','ou1337tmp');	
	
		byState:=	20;
		
	20:	CASE diResultStartOpcUa  OF

			0:	byState	:=	30;	//The OPC UA server is started.
			           	
			1:	byState	:=	31;	//The standard- user name and password is active.
									//Standard user name: Schneider
									//Standard password: ou1337tmp
									
			-1:	byState	:=	32;	//The OPC UA server is already running.				
	                   	
			-4:	byState	:=	33;	//An invalid combination of username and password e.g. one part empty.
								//The standard- user name and password is used. Standard user name: Schneider. Standard password: ou1337tmp
		END_CASE					
		
END_CASE

// ---------------------------- STOP OPC UA SERVER ----------------------------------
IF xStartUaServer = FALSE AND byState > 0 THEN
	
		diAddOverrunTime := 500 ;
		diAddWDogTime := 2000;
		
		SystemInterface.FC_CycleCheckTimeGet(iq_diOverrunTime := diOverrunTime, iq_diWDogFactor := diWDogTime);
		// Only call once when the server is stopped
		IF xCallOnceWhenStopServer THEN
			SystemInterface.FC_CycleCheckTimeSet(i_diOverrunTime := (diOverrunTime + diAddOverrunTime), i_diWDogFactor := (diWDogTime + diAddWDogTime));
			xCallOnceWhenStopServer := FALSE;
		END_IF
		
		diAddOverrunTimeSum := diAddOverrunTimeSum + diAddOverrunTime;
		diAddWDogTimeSum := diAddWDogTimeSum + diAddWDogTime;
		
		// Stop OPC UA Server	
		diResultStopOpcUa := SystemInterface.FC_OpcUaStop();
		
		byState:=	5;
END_IF	

// -------------------------------UA Diagnostic------------------------------
SystemInterface.FC_OpcUaGetServerConfig(iq_stOpcUaServerConfig	:= stOpcUaServerConfig);

END_PROGRAM

// LMC_PacDrive/Application/TemplateFullProgrammingFramework/TaskCalls/SR_MainMachine
PROGRAM  SR_MainMachine
VAR CONSTANT
	c_udiNumberOfGroups			: UDINT := 3;		(* Maximum number of groups *)
	c_udiNumberOfGroupMembers	: UDINT := 3;		(* Maximum number of members per group *)

	c_udiNumberOfCmdTables		: UDINT := 14;		(* Must be the exact number of used CMDTables! *)
	c_udiNumberOfCmdSteps		: UDINT := 16;		(* Make sure that the number of command steps that each table
													   contains does not exceed the c_udiNumberOfCmdSteps variable.*)

(* Definition group of modules *)
	c_udiMasterGroup			: UDINT := 2001;	(* Name of module group  1 *)
	c_udiServoDrivesGroup		: UDINT := 2002;	(* Name of module group  2 *)

(* ModuleId of MainMachine *)
	c_udiMainModuleId			: UDINT := 1;		(* ModuleId *)

(* System generated code, could be modified for your application *)
	c_udiNumberOfSubModules		: UDINT := 3;		(* Number of SubModules *)
	c_udiAlpha					: UDINT := 1;		(* Name & number of Module 1 *)
	c_udiBravo					: UDINT := 2;		(* Name & number of Module 2 *)
	c_udiMultiCarrier			: UDINT := 3;		(* Name & number of Module 4 *)

	c_dwModuleType				: DWORD := TPL.ET_ModuleType.MachineModule;
	c_sModuleTypeName			: STRING[14] := 'MainMachine';
	c_udiModuleVersion			: UDINT := 1;
(* End of system generated code, could be modified for your application *)
END_VAR

VAR (* User specific variables *)
	xError					: BOOL;
	stMulticarrierModule	: ST_MulticarrierModule;
	iStateInitMultiCarrier	: INT;
	//--- Control Loop Parameter
	
	dwPosP_Straight			: DWORD;
	dwVelP_Straight			: DWORD;
	dwVelI_Straight			: DWORD;
	dwPosP_Curve			: DWORD;
	dwVelP_Curve			: DWORD;
	dwVelI_Curve			: DWORD;
	dwMaxCurr				: DWORD;
	dwMaxload				: DWORD;
	dwDeviationLevelWarning	: DWORD;
	dwDeviationLevelError	: DWORD;
END_VAR

VAR
	xInitSuccessful : BOOL;
		
(*INPUT Variables*)
	xInputErrorQuit				: BOOL;
	xInputStart					: BOOL;
	xInputStop					: BOOL;
	xInputPrepare				: BOOL;
	xInputAuto					: BOOL;
	xInputManual				: BOOL;
	xInputJogMachine			: BOOL;
	xInputHold					: BOOL;
	xInputAbort					: BOOL;
	xInputPowerOn				: BOOL;
	xInputPowerOff				: BOOL;
	xInputBrakeRelease			: BOOL;
	xInputTestMulticarrier		: BOOL;
	xInputTrackCalibration		: BOOL;
	xInputEmergency				: BOOL := TRUE;

(* OUTPUT Variables *)
	xOutputPrepareActive		: BOOL;
	xOutputAutoActive			: BOOL;
	xOutputHoldActive			: BOOL;
	xOutputServiceActive		: BOOL;
	xOutputManualActive			: BOOL;
	xOutputJogMachineActive		: BOOL;

(* User Exceptions declaration *)
	stSystemException1				: TPL.ST_Exception;
	stSystemException2				: TPL.ST_Exception;
	stSystemException3				: TPL.ST_Exception;
	
	stEmergencyStopException		: TPL.ST_Exception;
	stContactorControlException		: TPL.ST_Exception;
	
	stUpdateStructsException		: TPL.ST_Exception;
	xUpdateStructsException			: BOOL;
	
	stInitReactionsException		: TPL.ST_Exception;
	xInitReactionsException			: BOOL;
	
	stInitSubModulesException		: TPL.ST_Exception;
	xInitSubModulesException		: BOOL;
	
	stUserException1				: TPL.ST_Exception;
	stUserException2				: TPL.ST_Exception;
	stUserException3				: TPL.ST_Exception;
	stUserException4				: TPL.ST_Exception;
	stUserException5				: TPL.ST_Exception;

	etSetExceptionDiag1			: GD.ET_Diag;
	etSetExceptionDiag2			: GD.ET_Diag;
	etSetExceptionDiag3			: GD.ET_Diag;
	etSetExceptionDiag4			: GD.ET_Diag;
	etSetExceptionDiag5			: GD.ET_Diag;
	
	etSetExceptionDiagExt1		: TPL.ET_DiagExt;
	etSetExceptionDiagExt2		: TPL.ET_DiagExt;
	etSetExceptionDiagExt3		: TPL.ET_DiagExt;
	etSetExceptionDiagExt4		: TPL.ET_DiagExt;
	etSetExceptionDiagExt5		: TPL.ET_DiagExt;
	
	sSetExceptionMsg1			: STRING[80];
	sSetExceptionMsg2			: STRING[80];
	sSetExceptionMsg3			: STRING[80];
	sSetExceptionMsg4			: STRING[80];
	sSetExceptionMsg5			: STRING[80];

(* OPM control Variables *)
	xActPrepare					: BOOL;
	xActAuto					: BOOL;
	xActManual					: BOOL;
	xActJogMachine				: BOOL;
	xActBrake					: BOOL;
	xActTestMulticarrier		: BOOL;
	xActTrackCalibration		: BOOL;
	xCmdWasActive				: BOOL;

	xModeReady					: BOOL;
	xBrakeReady					: BOOL;
	xExitStop					: BOOL;

(* ApplicationLogger *)
	fbLoggerPoint					: APL.FB_LoggerPoint;
	
(* Main ModuleController *)
	fbModuleController				: TPL.FB_ModuleController;
	etDiagModuleController			: GD.ET_Diag;
	etDiagExtModuleController		: TPL.ET_DiagExt;
	sMsgModuleController			: STRING[80];
	xWaitForStartStep				: BOOL;

(* Standard related variables *)
	astSubModuleInterface		: ARRAY[1..c_udiNumberOfSubModules] OF TPL.ST_StandardModuleInterface;	(* Standard Module interface *)
	aaudiSubModuleGroups		: ARRAY[1..c_udiNumberOfGroups,1..c_udiNumberOfGroupMembers] OF UDINT;
	adwSubModuleAddInterfaces	: ARRAY[1..c_udiNumberOfSubModules] OF DWORD;
	
(* Machine interface *)
	stMachineInterface			: TPL.ST_StandardModuleInterface;
	stMachineMotionInterface	: TPL.ST_StandardMotionInterface;

(* Command table list *)
	astListofCMDTables			: ARRAY [1..c_udiNumberOfCmdTables] OF TPL.ST_CmdTable;   (* Cmd list of tables*)
	udiTableIndex				: UDINT;
	udiStepIndex				: UDINT;
	diStep						: DINT;
	
	astPrepareTable				: ARRAY [1..c_udiNumberOfCmdSteps] OF TPL.ST_Cmd; (* Relating  Cmd table *)
	astAutoTable				: ARRAY [1..c_udiNumberOfCmdSteps] OF TPL.ST_Cmd; (* Relating  Cmd table *)
	astManualTable				: ARRAY [1..c_udiNumberOfCmdSteps] OF TPL.ST_Cmd; (* Relating  Cmd table *)
	astHoldTable				: ARRAY [1..c_udiNumberOfCmdSteps] OF TPL.ST_Cmd; (* Relating  Cmd table *)
	astHoldJogMachineTable		: ARRAY [1..c_udiNumberOfCmdSteps] OF TPL.ST_Cmd; (* Relating  Cmd table *)
	astStartTable				: ARRAY [1..c_udiNumberOfCmdSteps] OF TPL.ST_Cmd; (* Relating  Cmd table *)
	astStopTable				: ARRAY [1..c_udiNumberOfCmdSteps] OF TPL.ST_Cmd; (* Relating  Cmd table *)
	astBrakeReleaseTable		: ARRAY [1..c_udiNumberOfCmdSteps] OF TPL.ST_Cmd; (* Relating  Cmd table *)
	astAbortTable				: ARRAY [1..c_udiNumberOfCmdSteps] OF TPL.ST_Cmd; (* Relating  Cmd table *)
	astJogMachineTable			: ARRAY [1..c_udiNumberOfCmdSteps] OF TPL.ST_Cmd; (* Relating  Cmd table *)
	astTestMulticarrierTable	: ARRAY [1..c_udiNumberOfCmdSteps] OF TPL.ST_Cmd; (* Relating  Cmd table *)
	astTrackCalibrationTable	: ARRAY [1..c_udiNumberOfCmdSteps] OF TPL.ST_Cmd; (* Relating  Cmd table *)
	astStopPrepareTable			: ARRAY [1..c_udiNumberOfCmdSteps] OF TPL.ST_Cmd; (* Relating  Cmd table *)
	astStopAutoTable			: ARRAY [1..c_udiNumberOfCmdSteps] OF TPL.ST_Cmd; (* Relating  Cmd table *)

(* ExceptionHandling related variables *)
	fbExceptionHandler				: TPL.FB_ExceptionHandler2;

	aetReactionTranslationMode		: ARRAY[1..c_udiNumberOfSubModules] OF TPL.ET_ReactionTranslationMode;
	aastReactionTranslationTable	: ARRAY[1..c_udiNumberOfSubModules,1..TPL.Gc_udiMaxNumberOfReactions] OF TPL.ST_Reaction;
	astReactionTranslationJobs		: ARRAY[1..c_udiNumberOfSubModules] OF TPL.ST_ReactionTranslationJobs;

	xCheckExceptionList				: BOOL := TRUE;
	xReactionActive					: BOOL;
	xVirtualSystem					: BOOL;

(* Contactor Control related variables *)
	fbContactorControl			: TPL.FB_ContactorControl;
	xMainsOn					: BOOL := TRUE;
	xMainsWatch					: BOOL;
	timPowerOnDelay				: TIME := T#1S;

	xContactorControlActive				: BOOL;
	xContactorControlReady				: BOOL;
	etContactorControlDiag				: GD.ET_Diag;		
	etContactorControlDiagExt			: TPL.ET_DiagExt;
	sContactorControlMsg				: STRING[80];
	xContactorControlPowerOnDelayOver	: BOOL;

(* Logging related variables*)
	fbLogger					: TPL.FB_Logger;

(* OnlineChange related variables *)
	fbDetectOnlineChange			: TPL.FB_DetectOnlineChange;
	xDetectOnlineChangeActive		: BOOL; 
	xDetectOnlineChangeReady		: BOOL; 
	etDetectOnlineChangeDiag		: GD.ET_Diag;
	etDetectOnlineChangeDiagExt		: TPL.ET_DiagExt; 
	sDetectOnlineChangeMsg			: STRING[80];

(* Exception  *)
	xTestUserException1				: BOOL;
	xTestUserException2				: BOOL;
	xTestUserException3				: BOOL;
	xTestUserException4				: BOOL;
	xTestUserException5				: BOOL;

	iTemp						: INT;
	diClassTemp					: DINT;

	stDiagSource				: SystemConfiguration.ST_LogicalAddress;
	sInstanceName				: STRING[80];
	diDiagClass					: DINT;
	diDiagCode					: DINT;
	diDiagCode_old				: DINT;
	sDiagMsg					: STRING[40];
	sDiagMsgExt					: STRING[15];
	ifDiagnosis					: SystemConfigurationItf.IF_Diagnosis;
	xSuccess					: BOOL;
	
(* POU-Feedback related variables*)	
	etDiag			: GD.ET_Diag;
	etDiagExt		: ET_DiagExt;
	etDiagExtTPL	: TPL.ET_DiagExt;
	
(* Set Interfaces *)
	xSuccessSetTrackInterfaces	: BOOL;
	xSuccessSetSegmentInterfaces: BOOL;
	xSuccessSetCarrierInterfaces: BOOL;
END_VAR
VAR // added by the converter: edge detectors and wires of the graphical bodies
    _w1 : BOOL;
END_VAR

